LIN {X 0,Y 245.755,Z 1206.562,A -85,B 0,C 180,E1 11861.498,E2 11861.498} C_VEL
LIN {X 0,Y 251.212,Z 1202.888,A -85,B 0,C 180,E1 11857.29,E2 11857.29} C_VEL
LIN {X 0,Y 258.789,Z 1196.828,A -85,B 0,C 180,E1 11852.877,E2 11852.877} C_VEL
LIN {X 0,Y 267.973,Z 1188.669,A -85,B 0,C 180,E1 11848.76,E2 11848.76} C_VEL
LIN {X 0,Y 278.335,Z 1179.083,A -85,B 0,C 180,E1 11845.169,E2 11845.169} C_VEL
LIN {X 0,Y 289.084,Z 1169.149,A -85,B 0,C 180,E1 11842.216,E2 11842.216} C_VEL
LIN {X 0,Y 274.237,Z 1186.667,A -85,B 0,C 180,E1 11838.684,E2 11838.684} C_VEL
LIN {X 0,Y 269.596,Z 1192.92,A -85,B 0,C 180,E1 11837.251,E2 11837.251} C_VEL
LIN {X 0,Y 262.948,Z 1209.699,A -85,B 0,C 180,E1 11834.368,E2 11834.368} C_VEL
LIN {X 0,Y 256.592,Z 1224.704,A -85,B 0,C 180,E1 11831.19,E2 11831.19} C_VEL
LIN {X 0,Y 250.584,Z 1238.42,A -85,B 0,C 180,E1 11827.626,E2 11827.626} C_VEL
LIN {X 0,Y 244.864,Z 1251.431,A -85,B 0,C 180,E1 11823.454,E2 11823.454} C_VEL
LIN {X 0,Y 240.269,Z 1262.385,A -85,B 0,C 180,E1 11819.086,E2 11819.086} C_VEL
LIN {X 0,Y 236.737,Z 1271.709,A -85,B 0,C 180,E1 11814.451,E2 11814.451} C_VEL
LIN {X 0,Y 234.239,Z 1279.61,A -85,B 0,C 180,E1 11809.449,E2 11809.449} C_VEL
LIN {X 0,Y 232.909,Z 1285.561,A -85,B 0,C 180,E1 11804.419,E2 11804.419} C_VEL
LIN {X 0,Y 232.494,Z 1289.538,A -85,B 0,C 180,E1 11799.656,E2 11799.656} C_VEL
LIN {X 0,Y 232.55,Z 1291.91,A -85,B 0,C 180,E1 11795.181,E2 11795.181} C_VEL
LIN {X 0,Y 232.656,Z 1292.783,A -85,B 0,C 180,E1 11791.232,E2 11791.232} C_VEL
LIN {X 0,Y 232.611,Z 1292.569,A -85,B 0,C 180,E1 11787.044,E2 11787.044} C_VEL
LIN {X 0,Y 232.476,Z 1291.001,A -85,B 0,C 180,E1 11782.836,E2 11782.836} C_VEL
LIN {X 0,Y 232.564,Z 1287.833,A -85,B 0,C 180,E1 11778.092,E2 11778.092} C_VEL
LIN {X 0,Y 233.279,Z 1283.097,A -85,B 0,C 180,E1 11773.313,E2 11773.313} C_VEL
LIN {X 0,Y 235.041,Z 1276.237,A -85,B 0,C 180,E1 11768.28,E2 11768.28} C_VEL
LIN {X 0,Y 237.87,Z 1267.902,A -85,B 0,C 180,E1 11763.542,E2 11763.542} C_VEL
LIN {X 0,Y 241.926,Z 1257.624,A -85,B 0,C 180,E1 11758.896,E2 11758.896} C_VEL
LIN {X 0,Y 246.929,Z 1245.842,A -85,B 0,C 180,E1 11754.619,E2 11754.619} C_VEL
LIN {X 0,Y 252.321,Z 1233.449,A -85,B 0,C 180,E1 11750.947,E2 11750.947} C_VEL
LIN {X 0,Y 258.618,Z 1218.846,A -85,B 0,C 180,E1 11747.425,E2 11747.425} C_VEL
LIN {X 0,Y 265.286,Z 1202.614,A -85,B 0,C 180,E1 11744.268,E2 11744.268} C_VEL
LIN {X 0,Y 271.623,Z 1185.934,A -85,B 0,C 180,E1 11741.649,E2 11741.649} C_VEL
LIN {X 0,Y 277.349,Z 1169.272,A -85,B 0,C 180,E1 11739.515,E2 11739.515} C_VEL
LIN {X 0,Y 283.124,Z 1150.359,A -85,B 0,C 180,E1 11737.565,E2 11737.565} C_VEL
LIN {X 0,Y 288.024,Z 1131.481,A -85,B 0,C 180,E1 11736.019,E2 11736.019} C_VEL
LIN {X 0,Y 292.141,Z 1112.055,A -85,B 0,C 180,E1 11734.776,E2 11734.776} C_VEL
LIN {X 0,Y 295.622,Z 1090.355,A -85,B 0,C 180,E1 11733.771,E2 11733.771} C_VEL
LIN {X 0,Y 297.824,Z 1068.85,A -85,B 0,C 180,E1 11733.095,E2 11733.095} C_VEL
LIN {X 0,Y 300.881,Z 1025.521,A -85,B 0,C 180,E1 11732.117,E2 11732.117} C_VEL
LIN {X 0,Y 303.528,Z 1000.807,A -85,B 0,C 180,E1 11731.837,E2 11731.837} C_VEL
LIN {X 0,Y 305.997,Z 989.84,A -85,B 0,C 180,E1 11731.66,E2 11731.66} C_VEL
LIN {X 0,Y 318.999,Z 964.24,A -85,B 0,C 180,E1 11730.364,E2 11730.364} C_VEL
LIN {X 0,Y 315.803,Z 942.601,A -85,B 0,C 180,E1 11727.022,E2 11727.022} C_VEL
LIN {X 0,Y 315.15,Z 920.536,A -85,B 0,C 180,E1 11723.86,E2 11723.86} C_VEL
LIN {X 0,Y 316.957,Z 896.197,A -85,B 0,C 180,E1 11720.689,E2 11720.689} C_VEL
LIN {X 0,Y 321.01,Z 872.026,A -85,B 0,C 180,E1 11717.866,E2 11717.866} C_VEL
LIN {X 0,Y 322.933,Z 862.716,A -85,B 0,C 180,E1 11716.827,E2 11716.827} C_VEL
LIN {X 0,Y 315.425,Z 847.371,A -85,B 0,C 180,E1 11712.634,E2 11712.634} C_VEL
LIN {X 0,Y 308.32,Z 833.413,A -85,B 0,C 180,E1 11708.391,E2 11708.391} C_VEL
LIN {X 0,Y 302.039,Z 821.447,A -85,B 0,C 180,E1 11704.366,E2 11704.366} C_VEL
LIN {X 0,Y 295.476,Z 809.112,A -85,B 0,C 180,E1 11699.806,E2 11699.806} C_VEL
LIN {X 0,Y 289.595,Z 798.554,A -85,B 0,C 180,E1 11695.445,E2 11695.445} C_VEL
LIN {X 0,Y 285.543,Z 791.156,A -85,B 0,C 180,E1 11692.151,E2 11692.151} C_VEL
LIN {X 0,Y 289.879,Z 787.525,A -85,B 0,C 180,E1 11688.056,E2 11688.056} C_VEL
LIN {X 0,Y 293.724,Z 785.356,A -85,B 0,C 180,E1 11685.208,E2 11685.208} C_VEL
LIN {X 0,Y 295.4,Z 784.737,A -85,B 0,C 180,E1 11684.087,E2 11684.087} C_VEL
LIN {X 0,Y 298.61,Z 791.453,A -85,B 0,C 180,E1 11680.59,E2 11680.59} C_VEL
LIN {X 0,Y 303.9,Z 799.813,A -85,B 0,C 180,E1 11677.359,E2 11677.359} C_VEL
LIN {X 0,Y 310.112,Z 810.178,A -85,B 0,C 180,E1 11674.146,E2 11674.146} C_VEL
LIN {X 0,Y 316.83,Z 822.326,A -85,B 0,C 180,E1 11671.128,E2 11671.128} C_VEL
LIN {X 0,Y 322.139,Z 832.942,A -85,B 0,C 180,E1 11668.972,E2 11668.972} C_VEL
LIN {X 0,Y 306.661,Z 1049.725,A -85,B 0,C 180,E1 11664.3,E2 11664.3} C_VEL
LIN {X 0,Y 304.158,Z 1070.256,A -85,B 0,C 180,E1 11663.577,E2 11663.577} C_VEL
LIN {X 0,Y 300.574,Z 1090.531,A -85,B 0,C 180,E1 11662.568,E2 11662.568} C_VEL
LIN {X 0,Y 296.047,Z 1110.096,A -85,B 0,C 180,E1 11661.275,E2 11661.275} C_VEL
LIN {X 0,Y 290.869,Z 1128.33,A -85,B 0,C 180,E1 11659.739,E2 11659.739} C_VEL
LIN {X 0,Y 284.758,Z 1146.545,A -85,B 0,C 180,E1 11657.804,E2 11657.804} C_VEL
LIN {X 0,Y 278.126,Z 1163.631,A -85,B 0,C 180,E1 11655.527,E2 11655.527} C_VEL
LIN {X 0,Y 271.382,Z 1179.111,A -85,B 0,C 180,E1 11652.967,E2 11652.967} C_VEL
LIN {X 0,Y 264.466,Z 1193.663,A -85,B 0,C 180,E1 11649.993,E2 11649.993} C_VEL
LIN {X 0,Y 257.465,Z 1207.393,A -85,B 0,C 180,E1 11646.497,E2 11646.497} C_VEL
LIN {X 0,Y 250.894,Z 1219.705,A -85,B 0,C 180,E1 11642.546,E2 11642.546} C_VEL
LIN {X 0,Y 245.417,Z 1229.787,A -85,B 0,C 180,E1 11638.467,E2 11638.467} C_VEL
LIN {X 0,Y 240.745,Z 1238.513,A -85,B 0,C 180,E1 11633.977,E2 11633.977} C_VEL
LIN {X 0,Y 237.146,Z 1245.644,A -85,B 0,C 180,E1 11629.189,E2 11629.189} C_VEL
LIN {X 0,Y 234.629,Z 1251.19,A -85,B 0,C 180,E1 11624.057,E2 11624.057} C_VEL
LIN {X 0,Y 233.286,Z 1254.753,A -85,B 0,C 180,E1 11619.123,E2 11619.123} C_VEL
LIN {X 0,Y 232.704,Z 1256.778,A -85,B 0,C 180,E1 11614.188,E2 11614.188} C_VEL
LIN {X 0,Y 232.587,Z 1257.354,A -85,B 0,C 180,E1 11609.506,E2 11609.506} C_VEL
LIN {X 0,Y 232.77,Z 1256.558,A -85,B 0,C 180,E1 11604.824,E2 11604.824} C_VEL
LIN {X 0,Y 233.416,Z 1254.378,A -85,B 0,C 180,E1 11600.133,E2 11600.133} C_VEL
LIN {X 0,Y 234.984,Z 1250.341,A -85,B 0,C 180,E1 11594.955,E2 11594.955} C_VEL
LIN {X 0,Y 237.562,Z 1244.786,A -85,B 0,C 180,E1 11590.066,E2 11590.066} C_VEL
LIN {X 0,Y 241.366,Z 1237.412,A -85,B 0,C 180,E1 11585.266,E2 11585.266} C_VEL
LIN {X 0,Y 246.175,Z 1228.535,A -85,B 0,C 180,E1 11580.83,E2 11580.83} C_VEL
LIN {X 0,Y 252.162,Z 1217.537,A -85,B 0,C 180,E1 11576.553,E2 11576.553} C_VEL
LIN {X 0,Y 258.483,Z 1205.616,A -85,B 0,C 180,E1 11572.883,E2 11572.883} C_VEL
LIN {X 0,Y 265.231,Z 1192.273,A -85,B 0,C 180,E1 11569.578,E2 11569.578} C_VEL
LIN {X 0,Y 272.222,Z 1177.437,A -85,B 0,C 180,E1 11566.618,E2 11566.618} C_VEL
LIN {X 0,Y 279.281,Z 1160.958,A -85,B 0,C 180,E1 11563.977,E2 11563.977} C_VEL
LIN {X 0,Y 285.708,Z 1144.096,A -85,B 0,C 180,E1 11561.805,E2 11561.805} C_VEL
LIN {X 0,Y 291.587,Z 1126.39,A -85,B 0,C 180,E1 11559.968,E2 11559.968} C_VEL
LIN {X 0,Y 297.09,Z 1106.623,A -85,B 0,C 180,E1 11558.356,E2 11558.356} C_VEL
LIN {X 0,Y 301.475,Z 1086.784,A -85,B 0,C 180,E1 11557.11,E2 11557.11} C_VEL
LIN {X 0,Y 302.005,Z 1083.684,A -85,B 0,C 180,E1 11556.935,E2 11556.935} C_VEL
LIN {X 0,Y 296.347,Z 1090.87,A -85,B 0,C 180,E1 11556.189,E2 11556.189} C_VEL
LIN {X 0,Y 293.428,Z 1094.102,A -85,B 0,C 180,E1 11555.748,E2 11555.748} C_VEL
LIN {X 0,Y 287.309,Z 1102.337,A -85,B 0,C 180,E1 11555.045,E2 11555.045} C_VEL
LIN {X 0,Y 285.957,Z 1103.878,A -85,B 0,C 180,E1 11554.857,E2 11554.857} C_VEL
LIN {X 0,Y 279.453,Z 1111.591,A -85,B 0,C 180,E1 11553.999,E2 11553.999} C_VEL
LIN {X 0,Y 268.229,Z 1125.113,A -85,B 0,C 180,E1 11552.715,E2 11552.715} C_VEL
LIN {X 0,Y 264.784,Z 1128.644,A -85,B 0,C 180,E1 11552.213,E2 11552.213} C_VEL
LIN {X 0,Y 259.686,Z 1132.965,A -85,B 0,C 180,E1 11551.266,E2 11551.266} C_VEL
LIN {X 0,Y 255.075,Z 1135.823,A -85,B 0,C 180,E1 11550.116,E2 11550.116} C_VEL
LIN {X 0,Y 253.809,Z 1136.519,A -85,B 0,C 180,E1 11549.76,E2 11549.76} C_VEL
LIN {X 0,Y 249.389,Z 1139.988,A -85,B 0,C 180,E1 11548.758,E2 11548.758} C_VEL
LIN {X 0,Y 245.814,Z 1141.922,A -85,B 0,C 180,E1 11547.627,E2 11547.627} C_VEL
LIN {X 0,Y 244.729,Z 1142.395,A -85,B 0,C 180,E1 11547.232,E2 11547.232} C_VEL
LIN {X 0,Y 240.474,Z 1145.51,A -85,B 0,C 180,E1 11546.089,E2 11546.089} C_VEL
LIN {X 0,Y 238.016,Z 1146.572,A -85,B 0,C 180,E1 11545.106,E2 11545.106} C_VEL
LIN {X 0,Y 237.268,Z 1146.582,A -85,B 0,C 180,E1 11544.658,E2 11544.658} C_VEL
LIN {X 0,Y 234.207,Z 1160.293,A -85,B 0,C 180,E1 11541.277,E2 11541.277} C_VEL
LIN {X 0,Y 231.739,Z 1171.635,A -85,B 0,C 180,E1 11537.839,E2 11537.839} C_VEL
LIN {X 0,Y 229.663,Z 1182.256,A -85,B 0,C 180,E1 11533.854,E2 11533.854} C_VEL
LIN {X 0,Y 228.345,Z 1190.868,A -85,B 0,C 180,E1 11529.833,E2 11529.833} C_VEL
LIN {X 0,Y 227.639,Z 1198.409,A -85,B 0,C 180,E1 11525.293,E2 11525.293} C_VEL
LIN {X 0,Y 227.7,Z 1204.054,A -85,B 0,C 180,E1 11520.755,E2 11520.755} C_VEL
LIN {X 0,Y 228.533,Z 1208.064,A -85,B 0,C 180,E1 11515.986,E2 11515.986} C_VEL
LIN {X 0,Y 230.183,Z 1210.229,A -85,B 0,C 180,E1 11511.508,E2 11511.508} C_VEL
LIN {X 0,Y 233.338,Z 1210.736,A -85,B 0,C 180,E1 11506.369,E2 11506.369} C_VEL
LIN {X 0,Y 237.731,Z 1209.285,A -85,B 0,C 180,E1 11501.613,E2 11501.613} C_VEL
LIN {X 0,Y 243.617,Z 1206.041,A -85,B 0,C 180,E1 11497.052,E2 11497.052} C_VEL
LIN {X 0,Y 251.038,Z 1200.995,A -85,B 0,C 180,E1 11492.74,E2 11492.74} C_VEL
LIN {X 0,Y 259.977,Z 1194.181,A -85,B 0,C 180,E1 11488.722,E2 11488.722} C_VEL
LIN {X 0,Y 271.054,Z 1185.201,A -85,B 0,C 180,E1 11484.869,E2 11484.869} C_VEL
LIN {X 0,Y 279.911,Z 1178.049,A -85,B 0,C 180,E1 11482.384,E2 11482.384} C_VEL
LIN {X 0,Y 266.206,Z 1192.836,A -85,B 0,C 180,E1 11479.022,E2 11479.022} C_VEL
LIN {X 0,Y 261.249,Z 1199.161,A -85,B 0,C 180,E1 11477.456,E2 11477.456} C_VEL
LIN {X 0,Y 254.581,Z 1214.76,A -85,B 0,C 180,E1 11474.513,E2 11474.513} C_VEL
LIN {X 0,Y 247.632,Z 1230.01,A -85,B 0,C 180,E1 11470.971,E2 11470.971} C_VEL
LIN {X 0,Y 241.173,Z 1243.865,A -85,B 0,C 180,E1 11466.953,E2 11466.953} C_VEL
LIN {X 0,Y 235.919,Z 1255.286,A -85,B 0,C 180,E1 11462.854,E2 11462.854} C_VEL
LIN {X 0,Y 231.476,Z 1265.398,A -85,B 0,C 180,E1 11458.37,E2 11458.37} C_VEL
LIN {X 0,Y 227.935,Z 1274.476,A -85,B 0,C 180,E1 11453.254,E2 11453.254} C_VEL
LIN {X 0,Y 225.745,Z 1281.555,A -85,B 0,C 180,E1 11448.063,E2 11448.063} C_VEL
LIN {X 0,Y 224.733,Z 1286.663,A -85,B 0,C 180,E1 11443.007,E2 11443.007} C_VEL
LIN {X 0,Y 224.499,Z 1290.151,A -85,B 0,C 180,E1 11437.937,E2 11437.937} C_VEL
LIN {X 0,Y 224.622,Z 1291.82,A -85,B 0,C 180,E1 11433.574,E2 11433.574} C_VEL
LIN {X 0,Y 224.683,Z 1292.221,A -85,B 0,C 180,E1 11429.236,E2 11429.236} C_VEL
LIN {X 0,Y 224.57,Z 1291.442,A -85,B 0,C 180,E1 11425.148,E2 11425.148} C_VEL
LIN {X 0,Y 224.475,Z 1289.247,A -85,B 0,C 180,E1 11420.515,E2 11420.515} C_VEL
LIN {X 0,Y 224.833,Z 1285.436,A -85,B 0,C 180,E1 11415.581,E2 11415.581} C_VEL
LIN {X 0,Y 226.141,Z 1279.594,A -85,B 0,C 180,E1 11410.366,E2 11410.366} C_VEL
LIN {X 0,Y 228.519,Z 1272.303,A -85,B 0,C 180,E1 11405.44,E2 11405.44} C_VEL
LIN {X 0,Y 232.281,Z 1262.786,A -85,B 0,C 180,E1 11400.401,E2 11400.401} C_VEL
LIN {X 0,Y 237.232,Z 1251.545,A -85,B 0,C 180,E1 11395.697,E2 11395.697} C_VEL
LIN {X 0,Y 242.909,Z 1239.257,A -85,B 0,C 180,E1 11391.573,E2 11391.573} C_VEL
LIN {X 0,Y 249.126,Z 1225.826,A -85,B 0,C 180,E1 11387.915,E2 11387.915} C_VEL
LIN {X 0,Y 256.065,Z 1210.193,A -85,B 0,C 180,E1 11384.479,E2 11384.479} C_VEL
LIN {X 0,Y 263.051,Z 1193.366,A -85,B 0,C 180,E1 11381.515,E2 11381.515} C_VEL
LIN {X 0,Y 269.639,Z 1175.901,A -85,B 0,C 180,E1 11379.045,E2 11379.045} C_VEL
LIN {X 0,Y 275.69,Z 1157.961,A -85,B 0,C 180,E1 11377.016,E2 11377.016} C_VEL
LIN {X 0,Y 281.267,Z 1138.742,A -85,B 0,C 180,E1 11375.281,E2 11375.281} C_VEL
LIN {X 0,Y 286.067,Z 1118.874,A -85,B 0,C 180,E1 11373.892,E2 11373.892} C_VEL
LIN {X 0,Y 289.705,Z 1099.73,A -85,B 0,C 180,E1 11372.866,E2 11372.866} C_VEL
LIN {X 0,Y 292.638,Z 1078.212,A -85,B 0,C 180,E1 11372.055,E2 11372.055} C_VEL
LIN {X 0,Y 296.419,Z 1028.006,A -85,B 0,C 180,E1 11370.853,E2 11370.853} C_VEL
LIN {X 0,Y 299.151,Z 1002.191,A -85,B 0,C 180,E1 11370.546,E2 11370.546} C_VEL
LIN {X 0,Y 301.455,Z 986.208,A -85,B 0,C 180,E1 11370.504,E2 11370.504} C_VEL
LIN {X 0,Y 312.06,Z 965.62,A -85,B 0,C 180,E1 11369.46,E2 11369.46} C_VEL
LIN {X 0,Y 309.246,Z 943.916,A -85,B 0,C 180,E1 11366.085,E2 11366.085} C_VEL
LIN {X 0,Y 308.93,Z 921.474,A -85,B 0,C 180,E1 11362.853,E2 11362.853} C_VEL
LIN {X 0,Y 311.092,Z 897.155,A -85,B 0,C 180,E1 11359.662,E2 11359.662} C_VEL
LIN {X 0,Y 315.581,Z 872.382,A -85,B 0,C 180,E1 11356.757,E2 11356.757} C_VEL
LIN {X 0,Y 316.739,Z 866.806,A -85,B 0,C 180,E1 11356.128,E2 11356.128} C_VEL
LIN {X 0,Y 309.418,Z 851.782,A -85,B 0,C 180,E1 11351.935,E2 11351.935} C_VEL
LIN {X 0,Y 302.652,Z 838.342,A -85,B 0,C 180,E1 11347.784,E2 11347.784} C_VEL
LIN {X 0,Y 295.798,Z 825.23,A -85,B 0,C 180,E1 11343.294,E2 11343.294} C_VEL
LIN {X 0,Y 289.736,Z 813.938,A -85,B 0,C 180,E1 11339.011,E2 11339.011} C_VEL
LIN {X 0,Y 284.111,Z 803.743,A -85,B 0,C 180,E1 11334.75,E2 11334.75} C_VEL
LIN {X 0,Y 282.771,Z 801.018,A -85,B 0,C 180,E1 11333.503,E2 11333.503} C_VEL
LIN {X 0,Y 283.961,Z 799.112,A -85,B 0,C 180,E1 11331.903,E2 11331.903} C_VEL
LIN {X 0,Y 287.775,Z 795.306,A -85,B 0,C 180,E1 11327.967,E2 11327.967} C_VEL
LIN {X 0,Y 292.798,Z 792.422,A -85,B 0,C 180,E1 11324.146,E2 11324.146} C_VEL
LIN {X 0,Y 297.26,Z 799.603,A -85,B 0,C 180,E1 11320.753,E2 11320.753} C_VEL
LIN {X 0,Y 302.329,Z 807.848,A -85,B 0,C 180,E1 11317.594,E2 11317.594} C_VEL
LIN {X 0,Y 308.804,Z 819.094,A -85,B 0,C 180,E1 11314.183,E2 11314.183} C_VEL
LIN {X 0,Y 315.257,Z 831.409,A -85,B 0,C 180,E1 11311.23,E2 11311.23} C_VEL
LIN {X 0,Y 317.829,Z 836.982,A -85,B 0,C 180,E1 11310.13,E2 11310.13} C_VEL
LIN {X 0,Y 302.072,Z 1050.253,A -85,B 0,C 180,E1 11305.53,E2 11305.53} C_VEL
LIN {X 0,Y 299.478,Z 1070.877,A -85,B 0,C 180,E1 11304.803,E2 11304.803} C_VEL
LIN {X 0,Y 295.813,Z 1090.993,A -85,B 0,C 180,E1 11303.803,E2 11303.803} C_VEL
LIN {X 0,Y 291.448,Z 1109.477,A -85,B 0,C 180,E1 11302.594,E2 11302.594} C_VEL
LIN {X 0,Y 286.059,Z 1128.048,A -85,B 0,C 180,E1 11301.049,E2 11301.049} C_VEL
LIN {X 0,Y 279.744,Z 1146.295,A -85,B 0,C 180,E1 11299.122,E2 11299.122} C_VEL
LIN {X 0,Y 273.079,Z 1162.967,A -85,B 0,C 180,E1 11296.916,E2 11296.916} C_VEL
LIN {X 0,Y 266.054,Z 1178.641,A -85,B 0,C 180,E1 11294.346,E2 11294.346} C_VEL
LIN {X 0,Y 258.801,Z 1193.376,A -85,B 0,C 180,E1 11291.348,E2 11291.348} C_VEL
LIN {X 0,Y 251.787,Z 1206.637,A -85,B 0,C 180,E1 11287.988,E2 11287.988} C_VEL
LIN {X 0,Y 245.189,Z 1218.485,A -85,B 0,C 180,E1 11284.245,E2 11284.245} C_VEL
LIN {X 0,Y 239.22,Z 1228.924,A -85,B 0,C 180,E1 11280.095,E2 11280.095} C_VEL
LIN {X 0,Y 233.877,Z 1238.265,A -85,B 0,C 180,E1 11275.309,E2 11275.309} C_VEL
LIN {X 0,Y 229.869,Z 1245.584,A -85,B 0,C 180,E1 11270.362,E2 11270.362} C_VEL
LIN {X 0,Y 227.139,Z 1251.083,A -85,B 0,C 180,E1 11265.313,E2 11265.313} C_VEL
LIN {X 0,Y 225.519,Z 1254.938,A -85,B 0,C 180,E1 11260.177,E2 11260.177} C_VEL
LIN {X 0,Y 224.795,Z 1257.199,A -85,B 0,C 180,E1 11255.102,E2 11255.102} C_VEL
LIN {X 0,Y 224.614,Z 1257.974,A -85,B 0,C 180,E1 11250.254,E2 11250.254} C_VEL
LIN {X 0,Y 224.749,Z 1257.356,A -85,B 0,C 180,E1 11245.406,E2 11245.406} C_VEL
LIN {X 0,Y 225.409,Z 1255.288,A -85,B 0,C 180,E1 11240.295,E2 11240.295} C_VEL
LIN {X 0,Y 226.899,Z 1251.677,A -85,B 0,C 180,E1 11235.191,E2 11235.191} C_VEL
LIN {X 0,Y 229.493,Z 1246.383,A -85,B 0,C 180,E1 11230.132,E2 11230.132} C_VEL
LIN {X 0,Y 233.349,Z 1239.248,A -85,B 0,C 180,E1 11225.17,E2 11225.17} C_VEL
LIN {X 0,Y 238.253,Z 1230.631,A -85,B 0,C 180,E1 11220.592,E2 11220.592} C_VEL
LIN {X 0,Y 244.021,Z 1220.598,A -85,B 0,C 180,E1 11216.415,E2 11216.415} C_VEL
LIN {X 0,Y 250.847,Z 1208.461,A -85,B 0,C 180,E1 11212.421,E2 11212.421} C_VEL
LIN {X 0,Y 257.77,Z 1195.572,A -85,B 0,C 180,E1 11209.039,E2 11209.039} C_VEL
LIN {X 0,Y 264.932,Z 1181.274,A -85,B 0,C 180,E1 11206.018,E2 11206.018} C_VEL
LIN {X 0,Y 272.164,Z 1165.428,A -85,B 0,C 180,E1 11203.33,E2 11203.33} C_VEL
LIN {X 0,Y 279.018,Z 1148.488,A -85,B 0,C 180,E1 11201.032,E2 11201.032} C_VEL
LIN {X 0,Y 285.174,Z 1131.023,A -85,B 0,C 180,E1 11199.132,E2 11199.132} C_VEL
LIN {X 0,Y 290.676,Z 1112.726,A -85,B 0,C 180,E1 11197.545,E2 11197.545} C_VEL
LIN {X 0,Y 293.476,Z 1101.734,A -85,B 0,C 180,E1 11196.746,E2 11196.746} C_VEL
LIN {X 0,Y 287.29,Z 1109.159,A -85,B 0,C 180,E1 11196.028,E2 11196.028} C_VEL
LIN {X 0,Y 281.413,Z 1114.592,A -85,B 0,C 180,E1 11195.141,E2 11195.141} C_VEL
LIN {X 0,Y 278.677,Z 1116.83,A -85,B 0,C 180,E1 11194.659,E2 11194.659} C_VEL
LIN {X 0,Y 272.945,Z 1122.529,A -85,B 0,C 180,E1 11193.836,E2 11193.836} C_VEL
LIN {X 0,Y 266.829,Z 1127.206,A -85,B 0,C 180,E1 11192.657,E2 11192.657} C_VEL
LIN {X 0,Y 264.784,Z 1128.644,A -85,B 0,C 180,E1 11192.213,E2 11192.213} C_VEL
LIN {X 0,Y 248.595,Z 1143.852,A -85,B 0,C 180,E1 11189.563,E2 11189.563} C_VEL
LIN {X 0,Y 242.304,Z 1148.962,A -85,B 0,C 180,E1 11188.267,E2 11188.267} C_VEL
LIN {X 0,Y 237.762,Z 1152.003,A -85,B 0,C 180,E1 11187.012,E2 11187.012} C_VEL
LIN {X 0,Y 234.032,Z 1153.609,A -85,B 0,C 180,E1 11185.564,E2 11185.564} C_VEL
LIN {X 0,Y 230.264,Z 1156.037,A -85,B 0,C 180,E1 11184.363,E2 11184.363} C_VEL
LIN {X 0,Y 227.939,Z 1156.895,A -85,B 0,C 180,E1 11183.253,E2 11183.253} C_VEL
LIN {X 0,Y 227.443,Z 1156.889,A -85,B 0,C 180,E1 11182.896,E2 11182.896} C_VEL
LIN {X 0,Y 224.582,Z 1169.354,A -85,B 0,C 180,E1 11179.236,E2 11179.236} C_VEL
LIN {X 0,Y 222.224,Z 1180.722,A -85,B 0,C 180,E1 11175.128,E2 11175.128} C_VEL
LIN {X 0,Y 220.675,Z 1189.9,A -85,B 0,C 180,E1 11170.971,E2 11170.971} C_VEL
LIN {X 0,Y 219.784,Z 1198.079,A -85,B 0,C 180,E1 11166.269,E2 11166.269} C_VEL
LIN {X 0,Y 219.688,Z 1203.942,A -85,B 0,C 180,E1 11161.826,E2 11161.826} C_VEL
LIN {X 0,Y 220.396,Z 1208.645,A -85,B 0,C 180,E1 11156.88,E2 11156.88} C_VEL
LIN {X 0,Y 221.938,Z 1211.401,A -85,B 0,C 180,E1 11152.233,E2 11152.233} C_VEL
LIN {X 0,Y 224.856,Z 1212.645,A -85,B 0,C 180,E1 11147.154,E2 11147.154} C_VEL
LIN {X 0,Y 229.413,Z 1211.937,A -85,B 0,C 180,E1 11141.975,E2 11141.975} C_VEL
LIN {X 0,Y 235.33,Z 1209.441,A -85,B 0,C 180,E1 11137.255,E2 11137.255} C_VEL
LIN {X 0,Y 242.832,Z 1205.233,A -85,B 0,C 180,E1 11132.804,E2 11132.804} C_VEL
LIN {X 0,Y 252.404,Z 1199.012,A -85,B 0,C 180,E1 11128.474,E2 11128.474} C_VEL
LIN {X 0,Y 263.734,Z 1191.052,A -85,B 0,C 180,E1 11124.547,E2 11124.547} C_VEL
LIN {X 0,Y 270.68,Z 1186.09,A -85,B 0,C 180,E1 11122.579,E2 11122.579} C_VEL
LIN {X 0,Y 255.559,Z 1201.341,A -85,B 0,C 180,E1 11118.609,E2 11118.609} C_VEL
LIN {X 0,Y 253.29,Z 1204.034,A -85,B 0,C 180,E1 11117.851,E2 11117.851} C_VEL
LIN {X 0,Y 246.121,Z 1219.662,A -85,B 0,C 180,E1 11114.654,E2 11114.654} C_VEL
LIN {X 0,Y 239.159,Z 1233.99,A -85,B 0,C 180,E1 11111.025,E2 11111.025} C_VEL
LIN {X 0,Y 232.795,Z 1246.848,A -85,B 0,C 180,E1 11106.964,E2 11106.964} C_VEL
LIN {X 0,Y 227.221,Z 1258.223,A -85,B 0,C 180,E1 11102.47,E2 11102.47} C_VEL
LIN {X 0,Y 222.879,Z 1267.655,A -85,B 0,C 180,E1 11097.812,E2 11097.812} C_VEL
LIN {X 0,Y 219.465,Z 1276.134,A -85,B 0,C 180,E1 11092.502,E2 11092.502} C_VEL
LIN {X 0,Y 217.521,Z 1282.414,A -85,B 0,C 180,E1 11087.385,E2 11087.385} C_VEL
LIN {X 0,Y 216.654,Z 1287.055,A -85,B 0,C 180,E1 11082.258,E2 11082.258} C_VEL
LIN {X 0,Y 216.525,Z 1290.031,A -85,B 0,C 180,E1 11077.163,E2 11077.163} C_VEL
LIN {X 0,Y 216.677,Z 1291.463,A -85,B 0,C 180,E1 11072.381,E2 11072.381} C_VEL
LIN {X 0,Y 216.694,Z 1291.538,A -85,B 0,C 180,E1 11068.415,E2 11068.415} C_VEL
LIN {X 0,Y 216.545,Z 1290.509,A -85,B 0,C 180,E1 11063.905,E2 11063.905} C_VEL
LIN {X 0,Y 216.522,Z 1287.938,A -85,B 0,C 180,E1 11059.088,E2 11059.088} C_VEL
LIN {X 0,Y 217.172,Z 1283.472,A -85,B 0,C 180,E1 11053.691,E2 11053.691} C_VEL
LIN {X 0,Y 218.822,Z 1277.583,A -85,B 0,C 180,E1 11048.56,E2 11048.56} C_VEL
LIN {X 0,Y 221.688,Z 1269.965,A -85,B 0,C 180,E1 11043.481,E2 11043.481} C_VEL
LIN {X 0,Y 225.887,Z 1260.408,A -85,B 0,C 180,E1 11038.514,E2 11038.514} C_VEL
LIN {X 0,Y 231.114,Z 1249.411,A -85,B 0,C 180,E1 11033.96,E2 11033.96} C_VEL
LIN {X 0,Y 237.173,Z 1237.034,A -85,B 0,C 180,E1 11029.835,E2 11029.835} C_VEL
LIN {X 0,Y 244.095,Z 1222.822,A -85,B 0,C 180,E1 11026.03,E2 11026.03} C_VEL
LIN {X 0,Y 250.929,Z 1208.145,A -85,B 0,C 180,E1 11022.849,E2 11022.849} C_VEL
LIN {X 0,Y 258.185,Z 1191.463,A -85,B 0,C 180,E1 11019.936,E2 11019.936} C_VEL
LIN {X 0,Y 265.137,Z 1173.722,A -85,B 0,C 180,E1 11017.458,E2 11017.458} C_VEL
LIN {X 0,Y 271.336,Z 1155.84,A -85,B 0,C 180,E1 11015.477,E2 11015.477} C_VEL
LIN {X 0,Y 276.859,Z 1137.34,A -85,B 0,C 180,E1 11013.838,E2 11013.838} C_VEL
LIN {X 0,Y 281.765,Z 1117.546,A -85,B 0,C 180,E1 11012.473,E2 11012.473} C_VEL
LIN {X 0,Y 285.557,Z 1098,A -85,B 0,C 180,E1 11011.447,E2 11011.447} C_VEL
LIN {X 0,Y 288.522,Z 1077.053,A -85,B 0,C 180,E1 11010.685,E2 11010.685} C_VEL
LIN {X 0,Y 292.421,Z 1027.207,A -85,B 0,C 180,E1 11009.501,E2 11009.501} C_VEL
LIN {X 0,Y 295.203,Z 1001.467,A -85,B 0,C 180,E1 11009.21,E2 11009.21} C_VEL
LIN {X 0,Y 298.349,Z 980.02,A -85,B 0,C 180,E1 11009.191,E2 11009.191} C_VEL
LIN {X 0,Y 305.184,Z 966.967,A -85,B 0,C 180,E1 11008.528,E2 11008.528} C_VEL
LIN {X 0,Y 302.698,Z 944.459,A -85,B 0,C 180,E1 11005.011,E2 11005.011} C_VEL
LIN {X 0,Y 302.828,Z 921.579,A -85,B 0,C 180,E1 11001.702,E2 11001.702} C_VEL
LIN {X 0,Y 305.389,Z 897.359,A -85,B 0,C 180,E1 10998.516,E2 10998.516} C_VEL
LIN {X 0,Y 310.452,Z 871.627,A -85,B 0,C 180,E1 10995.504,E2 10995.504} C_VEL
LIN {X 0,Y 310.409,Z 870.542,A -85,B 0,C 180,E1 10995.315,E2 10995.315} C_VEL
LIN {X 0,Y 303.091,Z 855.47,A -85,B 0,C 180,E1 10991.03,E2 10991.03} C_VEL
LIN {X 0,Y 296.007,Z 841.466,A -85,B 0,C 180,E1 10986.594,E2 10986.594} C_VEL
LIN {X 0,Y 289.742,Z 829.447,A -85,B 0,C 180,E1 10982.373,E2 10982.373} C_VEL
LIN {X 0,Y 283.201,Z 817.126,A -85,B 0,C 180,E1 10977.571,E2 10977.571} C_VEL
LIN {X 0,Y 280.57,Z 812.077,A -85,B 0,C 180,E1 10975.4,E2 10975.4} C_VEL
LIN {X 0,Y 281.665,Z 809.646,A -85,B 0,C 180,E1 10973.579,E2 10973.579} C_VEL
LIN {X 0,Y 282.321,Z 808.421,A -85,B 0,C 180,E1 10972.675,E2 10972.675} C_VEL
LIN {X 0,Y 284.364,Z 805.526,A -85,B 0,C 180,E1 10970.283,E2 10970.283} C_VEL
LIN {X 0,Y 289.692,Z 801.488,A -85,B 0,C 180,E1 10965.611,E2 10965.611} C_VEL
LIN {X 0,Y 291.684,Z 800.728,A -85,B 0,C 180,E1 10964.185,E2 10964.185} C_VEL
LIN {X 0,Y 296.053,Z 807.925,A -85,B 0,C 180,E1 10960.825,E2 10960.825} C_VEL
LIN {X 0,Y 300.914,Z 816.19,A -85,B 0,C 180,E1 10957.741,E2 10957.741} C_VEL
LIN {X 0,Y 307.095,Z 827.439,A -85,B 0,C 180,E1 10954.409,E2 10954.409} C_VEL
LIN {X 0,Y 313.612,Z 840.434,A -85,B 0,C 180,E1 10951.361,E2 10951.361} C_VEL
LIN {X 0,Y 299.561,Z 1026.455,A -85,B 0,C 180,E1 10947.372,E2 10947.372} C_VEL
LIN {X 0,Y 297.181,Z 1055.167,A -85,B 0,C 180,E1 10946.671,E2 10946.671} C_VEL
LIN {X 0,Y 294.185,Z 1076.304,A -85,B 0,C 180,E1 10945.865,E2 10945.865} C_VEL
LIN {X 0,Y 289.917,Z 1097.326,A -85,B 0,C 180,E1 10944.734,E2 10944.734} C_VEL
LIN {X 0,Y 284.649,Z 1117.223,A -85,B 0,C 180,E1 10943.31,E2 10943.31} C_VEL
LIN {X 0,Y 278.772,Z 1135.395,A -85,B 0,C 180,E1 10941.647,E2 10941.647} C_VEL
LIN {X 0,Y 272.202,Z 1152.766,A -85,B 0,C 180,E1 10939.656,E2 10939.656} C_VEL
LIN {X 0,Y 264.731,Z 1170.047,A -85,B 0,C 180,E1 10937.168,E2 10937.168} C_VEL
LIN {X 0,Y 257.019,Z 1185.941,A -85,B 0,C 180,E1 10934.291,E2 10934.291} C_VEL
LIN {X 0,Y 249.506,Z 1200.082,A -85,B 0,C 180,E1 10931.086,E2 10931.086} C_VEL
LIN {X 0,Y 242.512,Z 1212.421,A -85,B 0,C 180,E1 10927.602,E2 10927.602} C_VEL
LIN {X 0,Y 235.623,Z 1223.997,A -85,B 0,C 180,E1 10923.479,E2 10923.479} C_VEL
LIN {X 0,Y 229.483,Z 1234.081,A -85,B 0,C 180,E1 10918.864,E2 10918.864} C_VEL
LIN {X 0,Y 224.49,Z 1242.394,A -85,B 0,C 180,E1 10913.909,E2 10913.909} C_VEL
LIN {X 0,Y 220.827,Z 1248.88,A -85,B 0,C 180,E1 10908.751,E2 10908.751} C_VEL
LIN {X 0,Y 218.458,Z 1253.62,A -85,B 0,C 180,E1 10903.497,E2 10903.497} C_VEL
LIN {X 0,Y 217.174,Z 1256.767,A -85,B 0,C 180,E1 10898.167,E2 10898.167} C_VEL
LIN {X 0,Y 216.701,Z 1258.316,A -85,B 0,C 180,E1 10893.173,E2 10893.173} C_VEL
LIN {X 0,Y 216.64,Z 1258.486,A -85,B 0,C 180,E1 10888.412,E2 10888.412} C_VEL
LIN {X 0,Y 216.956,Z 1257.439,A -85,B 0,C 180,E1 10883.383,E2 10883.383} C_VEL
LIN {X 0,Y 217.954,Z 1254.857,A -85,B 0,C 180,E1 10878.085,E2 10878.085} C_VEL
LIN {X 0,Y 220.082,Z 1250.369,A -85,B 0,C 180,E1 10872.551,E2 10872.551} C_VEL
LIN {X 0,Y 223.393,Z 1244.335,A -85,B 0,C 180,E1 10867.36,E2 10867.36} C_VEL
LIN {X 0,Y 228.037,Z 1236.501,A -85,B 0,C 180,E1 10862.339,E2 10862.339} C_VEL
LIN {X 0,Y 233.806,Z 1227.021,A -85,B 0,C 180,E1 10857.685,E2 10857.685} C_VEL
LIN {X 0,Y 240.385,Z 1216.103,A -85,B 0,C 180,E1 10853.501,E2 10853.501} C_VEL
LIN {X 0,Y 247.568,Z 1203.716,A -85,B 0,C 180,E1 10849.743,E2 10849.743} C_VEL
LIN {X 0,Y 254.723,Z 1190.653,A -85,B 0,C 180,E1 10846.567,E2 10846.567} C_VEL
LIN {X 0,Y 262.361,Z 1175.401,A -85,B 0,C 180,E1 10843.606,E2 10843.606} C_VEL
LIN {X 0,Y 269.499,Z 1159.55,A -85,B 0,C 180,E1 10841.136,E2 10841.136} C_VEL
LIN {X 0,Y 276.154,Z 1142.924,A -85,B 0,C 180,E1 10839.05,E2 10839.05} C_VEL
LIN {X 0,Y 282.482,Z 1124.618,A -85,B 0,C 180,E1 10837.211,E2 10837.211} C_VEL
LIN {X 0,Y 284.393,Z 1118.317,A -85,B 0,C 180,E1 10836.643,E2 10836.643} C_VEL
LIN {X 0,Y 279.173,Z 1122.52,A -85,B 0,C 180,E1 10835.844,E2 10835.844} C_VEL
LIN {X 0,Y 272.497,Z 1128.728,A -85,B 0,C 180,E1 10834.918,E2 10834.918} C_VEL
LIN {X 0,Y 266.186,Z 1133.264,A -85,B 0,C 180,E1 10833.775,E2 10833.775} C_VEL
LIN {X 0,Y 263.831,Z 1134.97,A -85,B 0,C 180,E1 10833.334,E2 10833.334} C_VEL
LIN {X 0,Y 257.369,Z 1139.923,A -85,B 0,C 180,E1 10832.121,E2 10832.121} C_VEL
LIN {X 0,Y 251.893,Z 1143.176,A -85,B 0,C 180,E1 10830.801,E2 10830.801} C_VEL
LIN {X 0,Y 246.751,Z 1146.696,A -85,B 0,C 180,E1 10829.628,E2 10829.628} C_VEL
LIN {X 0,Y 242.304,Z 1148.962,A -85,B 0,C 180,E1 10828.267,E2 10828.267} C_VEL
LIN {X 0,Y 226.363,Z 1161.768,A -85,B 0,C 180,E1 10824.567,E2 10824.567} C_VEL
LIN {X 0,Y 221.381,Z 1165.109,A -85,B 0,C 180,E1 10822.938,E2 10822.938} C_VEL
LIN {X 0,Y 220.813,Z 1165.424,A -85,B 0,C 180,E1 10822.71,E2 10822.71} C_VEL
LIN {X 0,Y 218.084,Z 1166.441,A -85,B 0,C 180,E1 10821.236,E2 10821.236} C_VEL
LIN {X 0,Y 217.588,Z 1166.582,A -85,B 0,C 180,E1 10820.793,E2 10820.793} C_VEL
LIN {X 0,Y 214.94,Z 1178.633,A -85,B 0,C 180,E1 10816.608,E2 10816.608} C_VEL
LIN {X 0,Y 213.056,Z 1188.702,A -85,B 0,C 180,E1 10812.192,E2 10812.192} C_VEL
LIN {X 0,Y 211.988,Z 1197.104,A -85,B 0,C 180,E1 10807.589,E2 10807.589} C_VEL
LIN {X 0,Y 211.704,Z 1203.925,A -85,B 0,C 180,E1 10802.708,E2 10802.708} C_VEL
LIN {X 0,Y 212.262,Z 1208.996,A -85,B 0,C 180,E1 10797.841,E2 10797.841} C_VEL
LIN {X 0,Y 213.797,Z 1212.479,A -85,B 0,C 180,E1 10792.746,E2 10792.746} C_VEL
LIN {X 0,Y 216.529,Z 1214.297,A -85,B 0,C 180,E1 10787.737,E2 10787.737} C_VEL
LIN {X 0,Y 221.31,Z 1214.32,A -85,B 0,C 180,E1 10782.109,E2 10782.109} C_VEL
LIN {X 0,Y 228.036,Z 1212.232,A -85,B 0,C 180,E1 10776.758,E2 10776.758} C_VEL
LIN {X 0,Y 236.73,Z 1208.121,A -85,B 0,C 180,E1 10771.768,E2 10771.768} C_VEL
LIN {X 0,Y 247.91,Z 1201.771,A -85,B 0,C 180,E1 10767.012,E2 10767.012} C_VEL
LIN {X 0,Y 260.62,Z 1193.925,A -85,B 0,C 180,E1 10762.964,E2 10762.964} C_VEL
LIN {X 0,Y 261.257,Z 1193.555,A -85,B 0,C 180,E1 10762.754,E2 10762.754} C_VEL
LIN {X 0,Y 245.963,Z 1207.944,A -85,B 0,C 180,E1 10758.502,E2 10758.502} C_VEL
LIN {X 0,Y 243.729,Z 1211.915,A -85,B 0,C 180,E1 10757.598,E2 10757.598} C_VEL
LIN {X 0,Y 236.963,Z 1225.626,A -85,B 0,C 180,E1 10754.463,E2 10754.463} C_VEL
LIN {X 0,Y 229.624,Z 1239.697,A -85,B 0,C 180,E1 10750.452,E2 10750.452} C_VEL
LIN {X 0,Y 223.027,Z 1252.164,A -85,B 0,C 180,E1 10745.966,E2 10745.966} C_VEL
LIN {X 0,Y 217.729,Z 1262.532,A -85,B 0,C 180,E1 10741.261,E2 10741.261} C_VEL
LIN {X 0,Y 213.508,Z 1271.516,A -85,B 0,C 180,E1 10736.118,E2 10736.118} C_VEL
LIN {X 0,Y 210.555,Z 1279.014,A -85,B 0,C 180,E1 10730.574,E2 10730.574} C_VEL
LIN {X 0,Y 209.04,Z 1284.435,A -85,B 0,C 180,E1 10725.254,E2 10725.254} C_VEL
LIN {X 0,Y 208.532,Z 1288.202,A -85,B 0,C 180,E1 10719.941,E2 10719.941} C_VEL
LIN {X 0,Y 208.613,Z 1290.301,A -85,B 0,C 180,E1 10714.95,E2 10714.95} C_VEL
LIN {X 0,Y 208.731,Z 1291.029,A -85,B 0,C 180,E1 10710.55,E2 10710.55} C_VEL
LIN {X 0,Y 208.64,Z 1290.518,A -85,B 0,C 180,E1 10705.879,E2 10705.879} C_VEL
LIN {X 0,Y 208.492,Z 1288.78,A -85,B 0,C 180,E1 10701.174,E2 10701.174} C_VEL
LIN {X 0,Y 208.792,Z 1285.3,A -85,B 0,C 180,E1 10695.865,E2 10695.865} C_VEL
LIN {X 0,Y 210.114,Z 1279.943,A -85,B 0,C 180,E1 10690.255,E2 10690.255} C_VEL
LIN {X 0,Y 212.622,Z 1273.162,A -85,B 0,C 180,E1 10684.963,E2 10684.963} C_VEL
LIN {X 0,Y 216.709,Z 1264.059,A -85,B 0,C 180,E1 10679.503,E2 10679.503} C_VEL
LIN {X 0,Y 222.061,Z 1253.329,A -85,B 0,C 180,E1 10674.492,E2 10674.492} C_VEL
LIN {X 0,Y 228.458,Z 1241.04,A -85,B 0,C 180,E1 10669.959,E2 10669.959} C_VEL
LIN {X 0,Y 235.174,Z 1228.078,A -85,B 0,C 180,E1 10666.133,E2 10666.133} C_VEL
LIN {X 0,Y 242.532,Z 1213.328,A -85,B 0,C 180,E1 10662.62,E2 10662.62} C_VEL
LIN {X 0,Y 250.147,Z 1197.062,A -85,B 0,C 180,E1 10659.519,E2 10659.519} C_VEL
LIN {X 0,Y 257.231,Z 1180.542,A -85,B 0,C 180,E1 10656.988,E2 10656.988} C_VEL
LIN {X 0,Y 264.168,Z 1162.483,A -85,B 0,C 180,E1 10654.784,E2 10654.784} C_VEL
LIN {X 0,Y 270.657,Z 1142.775,A -85,B 0,C 180,E1 10652.891,E2 10652.891} C_VEL
LIN {X 0,Y 276.021,Z 1123.186,A -85,B 0,C 180,E1 10651.441,E2 10651.441} C_VEL
LIN {X 0,Y 280.193,Z 1104.197,A -85,B 0,C 180,E1 10650.371,E2 10650.371} C_VEL
LIN {X 0,Y 283.523,Z 1083.688,A -85,B 0,C 180,E1 10649.511,E2 10649.511} C_VEL
LIN {X 0,Y 285.869,Z 1061.14,A -85,B 0,C 180,E1 10648.885,E2 10648.885} C_VEL
LIN {X 0,Y 288.605,Z 1026.263,A -85,B 0,C 180,E1 10648.109,E2 10648.109} C_VEL
LIN {X 0,Y 291.428,Z 1000.677,A -85,B 0,C 180,E1 10647.838,E2 10647.838} C_VEL
LIN {X 0,Y 295.062,Z 975.189,A -85,B 0,C 180,E1 10647.87,E2 10647.87} C_VEL
LIN {X 0,Y 295.703,Z 973.327,A -85,B 0,C 180,E1 10647.848,E2 10647.848} C_VEL
LIN {X 0,Y 298.321,Z 968.249,A -85,B 0,C 180,E1 10647.584,E2 10647.584} C_VEL
LIN {X 0,Y 296.225,Z 945.529,A -85,B 0,C 180,E1 10643.999,E2 10643.999} C_VEL
LIN {X 0,Y 296.741,Z 922.305,A -85,B 0,C 180,E1 10640.616,E2 10640.616} C_VEL
LIN {X 0,Y 299.836,Z 896.845,A -85,B 0,C 180,E1 10637.264,E2 10637.264} C_VEL
LIN {X 0,Y 304.302,Z 874.838,A -85,B 0,C 180,E1 10634.655,E2 10634.655} C_VEL
LIN {X 0,Y 297.018,Z 859.748,A -85,B 0,C 180,E1 10630.277,E2 10630.277} C_VEL
LIN {X 0,Y 289.963,Z 845.713,A -85,B 0,C 180,E1 10625.739,E2 10625.739} C_VEL
LIN {X 0,Y 283.707,Z 833.722,A -85,B 0,C 180,E1 10621.413,E2 10621.413} C_VEL
LIN {X 0,Y 278.585,Z 823.764,A -85,B 0,C 180,E1 10617.428,E2 10617.428} C_VEL
LIN {X 0,Y 279.618,Z 820.316,A -85,B 0,C 180,E1 10615.231,E2 10615.231} C_VEL
LIN {X 0,Y 281.631,Z 816.122,A -85,B 0,C 180,E1 10612.246,E2 10612.246} C_VEL
LIN {X 0,Y 283.763,Z 813.228,A -85,B 0,C 180,E1 10609.852,E2 10609.852} C_VEL
LIN {X 0,Y 288.999,Z 809.367,A -85,B 0,C 180,E1 10605.37,E2 10605.37} C_VEL
LIN {X 0,Y 290.45,Z 808.928,A -85,B 0,C 180,E1 10604.321,E2 10604.321} C_VEL
LIN {X 0,Y 294.179,Z 815.186,A -85,B 0,C 180,E1 10601.368,E2 10601.368} C_VEL
LIN {X 0,Y 298.81,Z 823.368,A -85,B 0,C 180,E1 10598.299,E2 10598.299} C_VEL
LIN {X 0,Y 304.59,Z 834.232,A -85,B 0,C 180,E1 10595.05,E2 10595.05} C_VEL
LIN {X 0,Y 309.636,Z 844.747,A -85,B 0,C 180,E1 10592.547,E2 10592.547} C_VEL
LIN {X 0,Y 293.303,Z 1051.587,A -85,B 0,C 180,E1 10588.094,E2 10588.094} C_VEL
LIN {X 0,Y 290.56,Z 1072.062,A -85,B 0,C 180,E1 10587.373,E2 10587.373} C_VEL
LIN {X 0,Y 286.504,Z 1092.892,A -85,B 0,C 180,E1 10586.337,E2 10586.337} C_VEL
LIN {X 0,Y 281.347,Z 1112.963,A -85,B 0,C 180,E1 10584.998,E2 10584.998} C_VEL
LIN {X 0,Y 275.648,Z 1130.995,A -85,B 0,C 180,E1 10583.459,E2 10583.459} C_VEL
LIN {X 0,Y 269.196,Z 1148.348,A -85,B 0,C 180,E1 10581.599,E2 10581.599} C_VEL
LIN {X 0,Y 261.814,Z 1165.446,A -85,B 0,C 180,E1 10579.292,E2 10579.292} C_VEL
LIN {X 0,Y 254.257,Z 1180.936,A -85,B 0,C 180,E1 10576.676,E2 10576.676} C_VEL
LIN {X 0,Y 246.43,Z 1195.497,A -85,B 0,C 180,E1 10573.609,E2 10573.609} C_VEL
LIN {X 0,Y 238.817,Z 1208.61,A -85,B 0,C 180,E1 10570.146,E2 10570.146} C_VEL
LIN {X 0,Y 231.605,Z 1220.328,A -85,B 0,C 180,E1 10566.258,E2 10566.258} C_VEL
LIN {X 0,Y 225.042,Z 1230.65,A -85,B 0,C 180,E1 10561.917,E2 10561.917} C_VEL
LIN {X 0,Y 219.101,Z 1239.919,A -85,B 0,C 180,E1 10556.857,E2 10556.857} C_VEL
LIN {X 0,Y 214.423,Z 1247.481,A -85,B 0,C 180,E1 10551.327,E2 10551.327} C_VEL
LIN {X 0,Y 211.284,Z 1253.034,A -85,B 0,C 180,E1 10545.647,E2 10545.647} C_VEL
LIN {X 0,Y 209.564,Z 1256.59,A -85,B 0,C 180,E1 10540.167,E2 10540.167} C_VEL
LIN {X 0,Y 208.809,Z 1258.608,A -85,B 0,C 180,E1 10534.668,E2 10534.668} C_VEL
LIN {X 0,Y 208.656,Z 1259.18,A -85,B 0,C 180,E1 10529.45,E2 10529.45} C_VEL
LIN {X 0,Y 208.869,Z 1258.45,A -85,B 0,C 180,E1 10524.505,E2 10524.505} C_VEL
LIN {X 0,Y 209.73,Z 1256.214,A -85,B 0,C 180,E1 10519.006,E2 10519.006} C_VEL
LIN {X 0,Y 211.725,Z 1252.182,A -85,B 0,C 180,E1 10513.256,E2 10513.256} C_VEL
LIN {X 0,Y 214.931,Z 1246.629,A -85,B 0,C 180,E1 10507.863,E2 10507.863} C_VEL
LIN {X 0,Y 219.556,Z 1239.255,A -85,B 0,C 180,E1 10502.615,E2 10502.615} C_VEL
LIN {X 0,Y 225.291,Z 1230.375,A -85,B 0,C 180,E1 10497.82,E2 10497.82} C_VEL
LIN {X 0,Y 232.307,Z 1219.371,A -85,B 0,C 180,E1 10493.253,E2 10493.253} C_VEL
LIN {X 0,Y 239.617,Z 1207.442,A -85,B 0,C 180,E1 10489.386,E2 10489.386} C_VEL
LIN {X 0,Y 247.318,Z 1194.088,A -85,B 0,C 180,E1 10485.943,E2 10485.943} C_VEL
LIN {X 0,Y 255.222,Z 1179.24,A -85,B 0,C 180,E1 10482.895,E2 10482.895} C_VEL
LIN {X 0,Y 263.122,Z 1162.745,A -85,B 0,C 180,E1 10480.199,E2 10480.199} C_VEL
LIN {X 0,Y 270.273,Z 1145.864,A -85,B 0,C 180,E1 10478.002,E2 10478.002} C_VEL
LIN {X 0,Y 275.253,Z 1132.113,A -85,B 0,C 180,E1 10476.501,E2 10476.501} C_VEL
LIN {X 0,Y 267.842,Z 1137.747,A -85,B 0,C 180,E1 10475.354,E2 10475.354} C_VEL
LIN {X 0,Y 263.463,Z 1140.696,A -85,B 0,C 180,E1 10474.559,E2 10474.559} C_VEL
LIN {X 0,Y 256.475,Z 1145.683,A -85,B 0,C 180,E1 10473.346,E2 10473.346} C_VEL
LIN {X 0,Y 250.724,Z 1148.998,A -85,B 0,C 180,E1 10472.032,E2 10472.032} C_VEL
LIN {X 0,Y 244.725,Z 1152.885,A -85,B 0,C 180,E1 10470.711,E2 10470.711} C_VEL
LIN {X 0,Y 240.213,Z 1155.092,A -85,B 0,C 180,E1 10469.418,E2 10469.418} C_VEL
LIN {X 0,Y 234.748,Z 1158.379,A -85,B 0,C 180,E1 10467.939,E2 10467.939} C_VEL
LIN {X 0,Y 231.435,Z 1159.738,A -85,B 0,C 180,E1 10466.7,E2 10466.7} C_VEL
LIN {X 0,Y 227.057,Z 1162.377,A -85,B 0,C 180,E1 10465.287,E2 10465.287} C_VEL
LIN {X 0,Y 223.615,Z 1163.727,A -85,B 0,C 180,E1 10463.73,E2 10463.73} C_VEL
LIN {X 0,Y 220.813,Z 1165.424,A -85,B 0,C 180,E1 10462.71,E2 10462.71} C_VEL
LIN {X 0,Y 216.013,Z 1168.61,A -85,B 0,C 180,E1 10460.825,E2 10460.825} C_VEL
LIN {X 0,Y 210.005,Z 1173.502,A -85,B 0,C 180,E1 10459.024,E2 10459.024} C_VEL
LIN {X 0,Y 207.9,Z 1175.818,A -85,B 0,C 180,E1 10458.321,E2 10458.321} C_VEL
LIN {X 0,Y 207.746,Z 1176.232,A -85,B 0,C 180,E1 10458.166,E2 10458.166} C_VEL
LIN {X 0,Y 205.516,Z 1187.299,A -85,B 0,C 180,E1 10453.505,E2 10453.505} C_VEL
LIN {X 0,Y 204.268,Z 1195.823,A -85,B 0,C 180,E1 10449.012,E2 10449.012} C_VEL
LIN {X 0,Y 203.759,Z 1203.728,A -85,B 0,C 180,E1 10443.658,E2 10443.658} C_VEL
LIN {X 0,Y 204.188,Z 1209.313,A -85,B 0,C 180,E1 10438.598,E2 10438.598} C_VEL
LIN {X 0,Y 205.761,Z 1213.599,A -85,B 0,C 180,E1 10433.023,E2 10433.023} C_VEL
LIN {X 0,Y 208.699,Z 1215.915,A -85,B 0,C 180,E1 10427.55,E2 10427.55} C_VEL
LIN {X 0,Y 213.156,Z 1216.473,A -85,B 0,C 180,E1 10422.249,E2 10422.249} C_VEL
LIN {X 0,Y 219.647,Z 1215.238,A -85,B 0,C 180,E1 10416.954,E2 10416.954} C_VEL
LIN {X 0,Y 228.436,Z 1212.007,A -85,B 0,C 180,E1 10411.79,E2 10411.79} C_VEL
LIN {X 0,Y 239.763,Z 1206.653,A -85,B 0,C 180,E1 10406.887,E2 10406.887} C_VEL
LIN {X 0,Y 251.84,Z 1200.314,A -85,B 0,C 180,E1 10402.942,E2 10402.942} C_VEL
LIN {X 0,Y 237.346,Z 1213.025,A -85,B 0,C 180,E1 10398.716,E2 10398.716} C_VEL
LIN {X 0,Y 229.337,Z 1228.139,A -85,B 0,C 180,E1 10395.067,E2 10395.067} C_VEL
LIN {X 0,Y 222.08,Z 1241.25,A -85,B 0,C 180,E1 10391.098,E2 10391.098} C_VEL
LIN {X 0,Y 215.423,Z 1253.137,A -85,B 0,C 180,E1 10386.588,E2 10386.588} C_VEL
LIN {X 0,Y 209.821,Z 1263.502,A -85,B 0,C 180,E1 10381.614,E2 10381.614} C_VEL
LIN {X 0,Y 205.305,Z 1272.585,A -85,B 0,C 180,E1 10375.997,E2 10375.997} C_VEL
LIN {X 0,Y 202.379,Z 1279.673,A -85,B 0,C 180,E1 10370.234,E2 10370.234} C_VEL
LIN {X 0,Y 200.938,Z 1284.702,A -85,B 0,C 180,E1 10364.702,E2 10364.702} C_VEL
LIN {X 0,Y 200.528,Z 1288.186,A -85,B 0,C 180,E1 10359.163,E2 10359.163} C_VEL
LIN {X 0,Y 200.657,Z 1289.914,A -85,B 0,C 180,E1 10354.288,E2 10354.288} C_VEL
LIN {X 0,Y 200.758,Z 1290.441,A -85,B 0,C 180,E1 10349.716,E2 10349.716} C_VEL
LIN {X 0,Y 200.625,Z 1289.756,A -85,B 0,C 180,E1 10345.141,E2 10345.141} C_VEL
LIN {X 0,Y 200.512,Z 1287.735,A -85,B 0,C 180,E1 10339.95,E2 10339.95} C_VEL
LIN {X 0,Y 200.961,Z 1284.23,A -85,B 0,C 180,E1 10334.712,E2 10334.712} C_VEL
LIN {X 0,Y 202.584,Z 1278.66,A -85,B 0,C 180,E1 10328.876,E2 10328.876} C_VEL
LIN {X 0,Y 205.68,Z 1271.251,A -85,B 0,C 180,E1 10323.123,E2 10323.123} C_VEL
LIN {X 0,Y 210.106,Z 1262.353,A -85,B 0,C 180,E1 10317.794,E2 10317.794} C_VEL
LIN {X 0,Y 215.786,Z 1251.842,A -85,B 0,C 180,E1 10312.841,E2 10312.841} C_VEL
LIN {X 0,Y 222.819,Z 1239.173,A -85,B 0,C 180,E1 10308.149,E2 10308.149} C_VEL
LIN {X 0,Y 230.671,Z 1224.843,A -85,B 0,C 180,E1 10303.986,E2 10303.986} C_VEL
LIN {X 0,Y 238.442,Z 1209.862,A -85,B 0,C 180,E1 10300.538,E2 10300.538} C_VEL
LIN {X 0,Y 246.121,Z 1193.966,A -85,B 0,C 180,E1 10297.612,E2 10297.612} C_VEL
LIN {X 0,Y 253.577,Z 1176.947,A -85,B 0,C 180,E1 10295.1,E2 10295.1} C_VEL
LIN {X 0,Y 260.857,Z 1158.247,A -85,B 0,C 180,E1 10292.923,E2 10292.923} C_VEL
LIN {X 0,Y 267.107,Z 1139.536,A -85,B 0,C 180,E1 10291.205,E2 10291.205} C_VEL
LIN {X 0,Y 272.541,Z 1120.058,A -85,B 0,C 180,E1 10289.817,E2 10289.817} C_VEL
LIN {X 0,Y 276.941,Z 1099.738,A -85,B 0,C 180,E1 10288.722,E2 10288.722} C_VEL
LIN {X 0,Y 280.161,Z 1079.468,A -85,B 0,C 180,E1 10287.96,E2 10287.96} C_VEL
LIN {X 0,Y 282.712,Z 1052.344,A -85,B 0,C 180,E1 10287.258,E2 10287.258} C_VEL
LIN {X 0,Y 285.011,Z 1024.729,A -85,B 0,C 180,E1 10286.669,E2 10286.669} C_VEL
LIN {X 0,Y 288.148,Z 997.331,A -85,B 0,C 180,E1 10286.421,E2 10286.421} C_VEL
LIN {X 0,Y 292.08,Z 969.829,A -85,B 0,C 180,E1 10286.48,E2 10286.48} C_VEL
LIN {X 0,Y 290.641,Z 961.837,A -85,B 0,C 180,E1 10285.359,E2 10285.359} C_VEL
LIN {X 0,Y 289.817,Z 938.688,A -85,B 0,C 180,E1 10281.769,E2 10281.769} C_VEL
LIN {X 0,Y 291.65,Z 913.975,A -85,B 0,C 180,E1 10278.265,E2 10278.265} C_VEL
LIN {X 0,Y 295.862,Z 888.896,A -85,B 0,C 180,E1 10275.083,E2 10275.083} C_VEL
LIN {X 0,Y 298.089,Z 878.819,A -85,B 0,C 180,E1 10273.876,E2 10273.876} C_VEL
LIN {X 0,Y 290.937,Z 864.001,A -85,B 0,C 180,E1 10269.492,E2 10269.492} C_VEL
LIN {X 0,Y 283.904,Z 849.876,A -85,B 0,C 180,E1 10264.848,E2 10264.848} C_VEL
LIN {X 0,Y 277.114,Z 836.767,A -85,B 0,C 180,E1 10260,E2 10260} C_VEL
LIN {X 0,Y 276.92,Z 835.746,A -85,B 0,C 180,E1 10259.379,E2 10259.379} C_VEL
LIN {X 0,Y 277.975,Z 830.64,A -85,B 0,C 180,E1 10256.391,E2 10256.391} C_VEL
LIN {X 0,Y 279.297,Z 826.986,A -85,B 0,C 180,E1 10254.041,E2 10254.041} C_VEL
LIN {X 0,Y 281.122,Z 823.595,A -85,B 0,C 180,E1 10251.615,E2 10251.615} C_VEL
LIN {X 0,Y 283.176,Z 820.942,A -85,B 0,C 180,E1 10249.42,E2 10249.42} C_VEL
LIN {X 0,Y 288.574,Z 817.137,A -85,B 0,C 180,E1 10244.938,E2 10244.938} C_VEL
LIN {X 0,Y 289.223,Z 817.082,A -85,B 0,C 180,E1 10244.459,E2 10244.459} C_VEL
LIN {X 0,Y 292.78,Z 823.194,A -85,B 0,C 180,E1 10241.585,E2 10241.585} C_VEL
LIN {X 0,Y 298.072,Z 833.04,A -85,B 0,C 180,E1 10238.036,E2 10238.036} C_VEL
LIN {X 0,Y 303.532,Z 843.918,A -85,B 0,C 180,E1 10234.947,E2 10234.947} C_VEL
LIN {X 0,Y 305.729,Z 848.909,A -85,B 0,C 180,E1 10233.798,E2 10233.798} C_VEL
LIN {X 0,Y 289.157,Z 1052.175,A -85,B 0,C 180,E1 10229.435,E2 10229.435} C_VEL
LIN {X 0,Y 286.321,Z 1072.712,A -85,B 0,C 180,E1 10228.715,E2 10228.715} C_VEL
LIN {X 0,Y 282.307,Z 1092.824,A -85,B 0,C 180,E1 10227.724,E2 10227.724} C_VEL
LIN {X 0,Y 277.54,Z 1111.243,A -85,B 0,C 180,E1 10226.528,E2 10226.528} C_VEL
LIN {X 0,Y 271.611,Z 1129.834,A -85,B 0,C 180,E1 10224.99,E2 10224.99} C_VEL
LIN {X 0,Y 264.757,Z 1147.784,A -85,B 0,C 180,E1 10223.096,E2 10223.096} C_VEL
LIN {X 0,Y 257.538,Z 1164.102,A -85,B 0,C 180,E1 10220.937,E2 10220.937} C_VEL
LIN {X 0,Y 249.712,Z 1179.819,A -85,B 0,C 180,E1 10218.342,E2 10218.342} C_VEL
LIN {X 0,Y 241.183,Z 1195.21,A -85,B 0,C 180,E1 10215.144,E2 10215.144} C_VEL
LIN {X 0,Y 233.178,Z 1208.478,A -85,B 0,C 180,E1 10211.653,E2 10211.653} C_VEL
LIN {X 0,Y 225.559,Z 1220.331,A -85,B 0,C 180,E1 10207.713,E2 10207.713} C_VEL
LIN {X 0,Y 218.578,Z 1230.76,A -85,B 0,C 180,E1 10203.292,E2 10203.292} C_VEL
LIN {X 0,Y 212.197,Z 1240.116,A -85,B 0,C 180,E1 10198.11,E2 10198.11} C_VEL
LIN {X 0,Y 207.317,Z 1247.434,A -85,B 0,C 180,E1 10192.694,E2 10192.694} C_VEL
LIN {X 0,Y 203.919,Z 1252.929,A -85,B 0,C 180,E1 10187.108,E2 10187.108} C_VEL
LIN {X 0,Y 201.815,Z 1256.875,A -85,B 0,C 180,E1 10181.196,E2 10181.196} C_VEL
LIN {X 0,Y 200.893,Z 1259.092,A -85,B 0,C 180,E1 10175.425,E2 10175.425} C_VEL
LIN {X 0,Y 200.687,Z 1259.82,A -85,B 0,C 180,E1 10169.999,E2 10169.999} C_VEL
LIN {X 0,Y 200.891,Z 1259.112,A -85,B 0,C 180,E1 10164.523,E2 10164.523} C_VEL
LIN {X 0,Y 201.787,Z 1256.968,A -85,B 0,C 180,E1 10158.844,E2 10158.844} C_VEL
LIN {X 0,Y 203.795,Z 1253.202,A -85,B 0,C 180,E1 10153.081,E2 10153.081} C_VEL
LIN {X 0,Y 207.061,Z 1247.916,A -85,B 0,C 180,E1 10147.574,E2 10147.574} C_VEL
LIN {X 0,Y 211.845,Z 1240.706,A -85,B 0,C 180,E1 10142.142,E2 10142.142} C_VEL
LIN {X 0,Y 217.887,Z 1231.824,A -85,B 0,C 180,E1 10137.116,E2 10137.116} C_VEL
LIN {X 0,Y 224.624,Z 1221.82,A -85,B 0,C 180,E1 10132.743,E2 10132.743} C_VEL
LIN {X 0,Y 232.124,Z 1210.287,A -85,B 0,C 180,E1 10128.772,E2 10128.772} C_VEL
LIN {X 0,Y 240.027,Z 1197.388,A -85,B 0,C 180,E1 10125.251,E2 10125.251} C_VEL
LIN {X 0,Y 248.128,Z 1183.078,A -85,B 0,C 180,E1 10122.144,E2 10122.144} C_VEL
LIN {X 0,Y 256.231,Z 1167.219,A -85,B 0,C 180,E1 10119.408,E2 10119.408} C_VEL
LIN {X 0,Y 263.883,Z 1150.191,A -85,B 0,C 180,E1 10117.08,E2 10117.08} C_VEL
LIN {X 0,Y 266.261,Z 1144.17,A -85,B 0,C 180,E1 10116.36,E2 10116.36} C_VEL
LIN {X 0,Y 263.084,Z 1146.228,A -85,B 0,C 180,E1 10115.823,E2 10115.823} C_VEL
LIN {X 0,Y 255.502,Z 1151.436,A -85,B 0,C 180,E1 10114.572,E2 10114.572} C_VEL
LIN {X 0,Y 248.687,Z 1155.252,A -85,B 0,C 180,E1 10113.148,E2 10113.148} C_VEL
LIN {X 0,Y 241.904,Z 1159.294,A -85,B 0,C 180,E1 10111.664,E2 10111.664} C_VEL
LIN {X 0,Y 237.928,Z 1161.209,A -85,B 0,C 180,E1 10110.564,E2 10110.564} C_VEL
LIN {X 0,Y 231.659,Z 1164.633,A -85,B 0,C 180,E1 10108.908,E2 10108.908} C_VEL
LIN {X 0,Y 228.075,Z 1166.164,A -85,B 0,C 180,E1 10107.679,E2 10107.679} C_VEL
LIN {X 0,Y 223.115,Z 1168.776,A -85,B 0,C 180,E1 10106.052,E2 10106.052} C_VEL
LIN {X 0,Y 220.022,Z 1169.984,A -85,B 0,C 180,E1 10104.714,E2 10104.714} C_VEL
LIN {X 0,Y 216.082,Z 1172.096,A -85,B 0,C 180,E1 10103.161,E2 10103.161} C_VEL
LIN {X 0,Y 213.54,Z 1172.902,A -85,B 0,C 180,E1 10101.71,E2 10101.71} C_VEL
LIN {X 0,Y 209.95,Z 1174.88,A -85,B 0,C 180,E1 10100.054,E2 10100.054} C_VEL
LIN {X 0,Y 207.948,Z 1175.356,A -85,B 0,C 180,E1 10098.503,E2 10098.503} C_VEL
LIN {X 0,Y 207.746,Z 1176.232,A -85,B 0,C 180,E1 10098.166,E2 10098.166} C_VEL
LIN {X 0,Y 205.82,Z 1180.721,A -85,B 0,C 180,E1 10096.483,E2 10096.483} C_VEL
LIN {X 0,Y 198.046,Z 1191.175,A -85,B 0,C 180,E1 10092.126,E2 10092.126} C_VEL
LIN {X 0,Y 196.531,Z 1194.842,A -85,B 0,C 180,E1 10090.183,E2 10090.183} C_VEL
LIN {X 0,Y 195.827,Z 1202.941,A -85,B 0,C 180,E1 10084.98,E2 10084.98} C_VEL
LIN {X 0,Y 196.069,Z 1209.146,A -85,B 0,C 180,E1 10079.708,E2 10079.708} C_VEL
LIN {X 0,Y 197.38,Z 1213.953,A -85,B 0,C 180,E1 10074.186,E2 10074.186} C_VEL
LIN {X 0,Y 200.117,Z 1217.072,A -85,B 0,C 180,E1 10068.472,E2 10068.472} C_VEL
LIN {X 0,Y 204.449,Z 1218.424,A -85,B 0,C 180,E1 10062.937,E2 10062.937} C_VEL
LIN {X 0,Y 210.847,Z 1218.048,A -85,B 0,C 180,E1 10057.412,E2 10057.412} C_VEL
LIN {X 0,Y 220.08,Z 1215.613,A -85,B 0,C 180,E1 10051.805,E2 10051.805} C_VEL
LIN {X 0,Y 231.555,Z 1211.208,A -85,B 0,C 180,E1 10046.744,E2 10046.744} C_VEL
LIN {X 0,Y 242.226,Z 1206.499,A -85,B 0,C 180,E1 10043.118,E2 10043.118} C_VEL
LIN {X 0,Y 229.571,Z 1216.77,A -85,B 0,C 180,E1 10039.275,E2 10039.275} C_VEL
LIN {X 0,Y 221.862,Z 1230.435,A -85,B 0,C 180,E1 10035.772,E2 10035.772} C_VEL
LIN {X 0,Y 214.142,Z 1243.51,A -85,B 0,C 180,E1 10031.532,E2 10031.532} C_VEL
LIN {X 0,Y 207.198,Z 1255.134,A -85,B 0,C 180,E1 10026.755,E2 10026.755} C_VEL
LIN {X 0,Y 201.36,Z 1265.276,A -85,B 0,C 180,E1 10021.426,E2 10021.426} C_VEL
LIN {X 0,Y 196.91,Z 1273.871,A -85,B 0,C 180,E1 10015.571,E2 10015.571} C_VEL
LIN {X 0,Y 194.11,Z 1280.535,A -85,B 0,C 180,E1 10009.563,E2 10009.563} C_VEL
LIN {X 0,Y 192.785,Z 1285.399,A -85,B 0,C 180,E1 10003.498,E2 10003.498} C_VEL
LIN {X 0,Y 192.55,Z 1288.187,A -85,B 0,C 180,E1 9998.061,E2 9998.061} C_VEL
LIN {X 0,Y 192.72,Z 1289.607,A -85,B 0,C 180,E1 9992.975,E2 9992.975} C_VEL
LIN {X 0,Y 192.762,Z 1289.736,A -85,B 0,C 180,E1 9988.515,E2 9988.515} C_VEL
LIN {X 0,Y 192.587,Z 1288.839,A -85,B 0,C 180,E1 9983.742,E2 9983.742} C_VEL
LIN {X 0,Y 192.579,Z 1286.423,A -85,B 0,C 180,E1 9978.319,E2 9978.319} C_VEL
LIN {X 0,Y 193.383,Z 1282.404,A -85,B 0,C 180,E1 9972.551,E2 9972.551} C_VEL
LIN {X 0,Y 195.573,Z 1276.419,A -85,B 0,C 180,E1 9966.5,E2 9966.5} C_VEL
LIN {X 0,Y 199.386,Z 1268.484,A -85,B 0,C 180,E1 9960.566,E2 9960.566} C_VEL
LIN {X 0,Y 204.6,Z 1259.033,A -85,B 0,C 180,E1 9955.128,E2 9955.128} C_VEL
LIN {X 0,Y 211.133,Z 1247.86,A -85,B 0,C 180,E1 9950.1,E2 9950.1} C_VEL
LIN {X 0,Y 218.617,Z 1235.13,A -85,B 0,C 180,E1 9945.595,E2 9945.595} C_VEL
LIN {X 0,Y 226.737,Z 1220.923,A -85,B 0,C 180,E1 9941.632,E2 9941.632} C_VEL
LIN {X 0,Y 234.976,Z 1205.695,A -85,B 0,C 180,E1 9938.274,E2 9938.274} C_VEL
LIN {X 0,Y 242.988,Z 1189.593,A -85,B 0,C 180,E1 9935.441,E2 9935.441} C_VEL
LIN {X 0,Y 250.569,Z 1172.615,A -85,B 0,C 180,E1 9933.075,E2 9933.075} C_VEL
LIN {X 0,Y 257.665,Z 1154.489,A -85,B 0,C 180,E1 9931.07,E2 9931.07} C_VEL
LIN {X 0,Y 264.004,Z 1135.536,A -85,B 0,C 180,E1 9929.419,E2 9929.419} C_VEL
LIN {X 0,Y 269.621,Z 1115.042,A -85,B 0,C 180,E1 9928.045,E2 9928.045} C_VEL
LIN {X 0,Y 274.047,Z 1094.235,A -85,B 0,C 180,E1 9927.028,E2 9927.028} C_VEL
LIN {X 0,Y 277.098,Z 1073.895,A -85,B 0,C 180,E1 9926.325,E2 9926.325} C_VEL
LIN {X 0,Y 281.182,Z 1027.521,A -85,B 0,C 180,E1 9925.263,E2 9925.263} C_VEL
LIN {X 0,Y 284.147,Z 1001.042,A -85,B 0,C 180,E1 9924.995,E2 9924.995} C_VEL
LIN {X 0,Y 287.868,Z 974.576,A -85,B 0,C 180,E1 9925.048,E2 9925.048} C_VEL
LIN {X 0,Y 288.196,Z 972.014,A -85,B 0,C 180,E1 9925.04,E2 9925.04} C_VEL
LIN {X 0,Y 284.365,Z 949.717,A -85,B 0,C 180,E1 9921.964,E2 9921.964} C_VEL
LIN {X 0,Y 283.523,Z 940.155,A -85,B 0,C 180,E1 9920.768,E2 9920.768} C_VEL
LIN {X 0,Y 285.71,Z 915.101,A -85,B 0,C 180,E1 9917.184,E2 9917.184} C_VEL
LIN {X 0,Y 290.283,Z 889.796,A -85,B 0,C 180,E1 9913.952,E2 9913.952} C_VEL
LIN {X 0,Y 291.857,Z 882.829,A -85,B 0,C 180,E1 9913.118,E2 9913.118} C_VEL
LIN {X 0,Y 284.55,Z 867.546,A -85,B 0,C 180,E1 9908.486,E2 9908.486} C_VEL
LIN {X 0,Y 277.774,Z 854.025,A -85,B 0,C 180,E1 9903.921,E2 9903.921} C_VEL
LIN {X 0,Y 275.521,Z 849.444,A -85,B 0,C 180,E1 9902.183,E2 9902.183} C_VEL
LIN {X 0,Y 275.867,Z 844.315,A -85,B 0,C 180,E1 9899.48,E2 9899.48} C_VEL
LIN {X 0,Y 277.3,Z 837.924,A -85,B 0,C 180,E1 9895.657,E2 9895.657} C_VEL
LIN {X 0,Y 278.694,Z 834.432,A -85,B 0,C 180,E1 9893.407,E2 9893.407} C_VEL
LIN {X 0,Y 280.56,Z 831.166,A -85,B 0,C 180,E1 9891.081,E2 9891.081} C_VEL
LIN {X 0,Y 282.606,Z 828.658,A -85,B 0,C 180,E1 9888.985,E2 9888.985} C_VEL
LIN {X 0,Y 287.895,Z 825.018,A -85,B 0,C 180,E1 9884.695,E2 9884.695} C_VEL
LIN {X 0,Y 291.249,Z 831.072,A -85,B 0,C 180,E1 9881.899,E2 9881.899} C_VEL
LIN {X 0,Y 295.91,Z 840.078,A -85,B 0,C 180,E1 9878.649,E2 9878.649} C_VEL
LIN {X 0,Y 301.015,Z 850.629,A -85,B 0,C 180,E1 9875.624,E2 9875.624} C_VEL
LIN {X 0,Y 301.973,Z 853.049,A -85,B 0,C 180,E1 9875.081,E2 9875.081} C_VEL
LIN {X 0,Y 285.167,Z 1052.829,A -85,B 0,C 180,E1 9870.812,E2 9870.812} C_VEL
LIN {X 0,Y 282.246,Z 1073.344,A -85,B 0,C 180,E1 9870.097,E2 9870.097} C_VEL
LIN {X 0,Y 278.125,Z 1093.402,A -85,B 0,C 180,E1 9869.114,E2 9869.114} C_VEL
LIN {X 0,Y 273.214,Z 1111.832,A -85,B 0,C 180,E1 9867.926,E2 9867.926} C_VEL
LIN {X 0,Y 267.102,Z 1130.429,A -85,B 0,C 180,E1 9866.395,E2 9866.395} C_VEL
LIN {X 0,Y 259.994,Z 1148.459,A -85,B 0,C 180,E1 9864.5,E2 9864.5} C_VEL
LIN {X 0,Y 252.555,Z 1164.707,A -85,B 0,C 180,E1 9862.352,E2 9862.352} C_VEL
LIN {X 0,Y 244.35,Z 1180.595,A -85,B 0,C 180,E1 9859.72,E2 9859.72} C_VEL
LIN {X 0,Y 235.571,Z 1195.821,A -85,B 0,C 180,E1 9856.533,E2 9856.533} C_VEL
LIN {X 0,Y 227.21,Z 1209.092,A -85,B 0,C 180,E1 9853.006,E2 9853.006} C_VEL
LIN {X 0,Y 219.222,Z 1220.946,A -85,B 0,C 180,E1 9849.005,E2 9849.005} C_VEL
LIN {X 0,Y 211.865,Z 1231.376,A -85,B 0,C 180,E1 9844.492,E2 9844.492} C_VEL
LIN {X 0,Y 205.1,Z 1240.733,A -85,B 0,C 180,E1 9839.175,E2 9839.175} C_VEL
LIN {X 0,Y 199.888,Z 1248.051,A -85,B 0,C 180,E1 9833.587,E2 9833.587} C_VEL
LIN {X 0,Y 196.228,Z 1253.545,A -85,B 0,C 180,E1 9827.8,E2 9827.8} C_VEL
LIN {X 0,Y 194.013,Z 1257.368,A -85,B 0,C 180,E1 9821.895,E2 9821.895} C_VEL
LIN {X 0,Y 192.966,Z 1259.64,A -85,B 0,C 180,E1 9815.947,E2 9815.947} C_VEL
LIN {X 0,Y 192.704,Z 1260.387,A -85,B 0,C 180,E1 9810.593,E2 9810.593} C_VEL
LIN {X 0,Y 192.878,Z 1259.857,A -85,B 0,C 180,E1 9804.943,E2 9804.943} C_VEL
LIN {X 0,Y 193.77,Z 1257.885,A -85,B 0,C 180,E1 9798.992,E2 9798.992} C_VEL
LIN {X 0,Y 195.784,Z 1254.37,A -85,B 0,C 180,E1 9793.075,E2 9793.075} C_VEL
LIN {X 0,Y 199.4,Z 1248.842,A -85,B 0,C 180,E1 9786.975,E2 9786.975} C_VEL
LIN {X 0,Y 204.432,Z 1241.706,A -85,B 0,C 180,E1 9781.359,E2 9781.359} C_VEL
LIN {X 0,Y 210.656,Z 1233.085,A -85,B 0,C 180,E1 9776.265,E2 9776.265} C_VEL
LIN {X 0,Y 217.812,Z 1223.045,A -85,B 0,C 180,E1 9771.704,E2 9771.704} C_VEL
LIN {X 0,Y 226.115,Z 1210.895,A -85,B 0,C 180,E1 9767.424,E2 9767.424} C_VEL
LIN {X 0,Y 234.371,Z 1197.994,A -85,B 0,C 180,E1 9763.863,E2 9763.863} C_VEL
LIN {X 0,Y 242.803,Z 1183.68,A -85,B 0,C 180,E1 9760.736,E2 9760.736} C_VEL
LIN {X 0,Y 251.207,Z 1167.817,A -85,B 0,C 180,E1 9757.992,E2 9757.992} C_VEL
LIN {X 0,Y 256.972,Z 1155.533,A -85,B 0,C 180,E1 9756.259,E2 9756.259} C_VEL
LIN {X 0,Y 249.083,Z 1159.948,A -85,B 0,C 180,E1 9754.752,E2 9754.752} C_VEL
LIN {X 0,Y 240.406,Z 1164.814,A -85,B 0,C 180,E1 9753.014,E2 9753.014} C_VEL
LIN {X 0,Y 234.763,Z 1167.543,A -85,B 0,C 180,E1 9751.59,E2 9751.59} C_VEL
LIN {X 0,Y 228.243,Z 1170.869,A -85,B 0,C 180,E1 9749.844,E2 9749.844} C_VEL
LIN {X 0,Y 224.737,Z 1172.355,A -85,B 0,C 180,E1 9748.718,E2 9748.718} C_VEL
LIN {X 0,Y 219.088,Z 1175.006,A -85,B 0,C 180,E1 9746.861,E2 9746.861} C_VEL
LIN {X 0,Y 216.366,Z 1176.059,A -85,B 0,C 180,E1 9745.747,E2 9745.747} C_VEL
LIN {X 0,Y 211.824,Z 1178.223,A -85,B 0,C 180,E1 9743.951,E2 9743.951} C_VEL
LIN {X 0,Y 209.015,Z 1179.251,A -85,B 0,C 180,E1 9742.501,E2 9742.501} C_VEL
LIN {X 0,Y 205.091,Z 1181.129,A -85,B 0,C 180,E1 9740.55,E2 9740.55} C_VEL
LIN {X 0,Y 203.268,Z 1181.657,A -85,B 0,C 180,E1 9739.243,E2 9739.243} C_VEL
LIN {X 0,Y 199.794,Z 1183.486,A -85,B 0,C 180,E1 9737.174,E2 9737.174} C_VEL
LIN {X 0,Y 198.42,Z 1183.79,A -85,B 0,C 180,E1 9735.743,E2 9735.743} C_VEL
LIN {X 0,Y 196.692,Z 1193.705,A -85,B 0,C 180,E1 9730.842,E2 9730.842} C_VEL
LIN {X 0,Y 196.531,Z 1194.842,A -85,B 0,C 180,E1 9730.183,E2 9730.183} C_VEL
LIN {X 0,Y 195.162,Z 1198.3,A -85,B 0,C 180,E1 9728.188,E2 9728.188} C_VEL
LIN {X 0,Y 190.063,Z 1204.601,A -85,B 0,C 180,E1 9724.193,E2 9724.193} C_VEL
LIN {X 0,Y 188.126,Z 1207.818,A -85,B 0,C 180,E1 9721.729,E2 9721.729} C_VEL
LIN {X 0,Y 187.993,Z 1208.895,A -85,B 0,C 180,E1 9720.767,E2 9720.767} C_VEL
LIN {X 0,Y 189.108,Z 1214.205,A -85,B 0,C 180,E1 9715.148,E2 9715.148} C_VEL
LIN {X 0,Y 191.877,Z 1218.192,A -85,B 0,C 180,E1 9708.884,E2 9708.884} C_VEL
LIN {X 0,Y 196.218,Z 1220.146,A -85,B 0,C 180,E1 9703.116,E2 9703.116} C_VEL
LIN {X 0,Y 202.699,Z 1220.449,A -85,B 0,C 180,E1 9697.372,E2 9697.372} C_VEL
LIN {X 0,Y 211.647,Z 1218.911,A -85,B 0,C 180,E1 9691.809,E2 9691.809} C_VEL
LIN {X 0,Y 223.831,Z 1215.249,A -85,B 0,C 180,E1 9686.365,E2 9686.365} C_VEL
LIN {X 0,Y 232.663,Z 1212.024,A -85,B 0,C 180,E1 9683.321,E2 9683.321} C_VEL
LIN {X 0,Y 221.734,Z 1220.527,A -85,B 0,C 180,E1 9679.848,E2 9679.848} C_VEL
LIN {X 0,Y 213.109,Z 1234.642,A -85,B 0,C 180,E1 9675.878,E2 9675.878} C_VEL
LIN {X 0,Y 204.923,Z 1247.64,A -85,B 0,C 180,E1 9671.201,E2 9671.201} C_VEL
LIN {X 0,Y 197.958,Z 1258.698,A -85,B 0,C 180,E1 9666.087,E2 9666.087} C_VEL
LIN {X 0,Y 192.396,Z 1267.916,A -85,B 0,C 180,E1 9660.618,E2 9660.618} C_VEL
LIN {X 0,Y 188.16,Z 1275.833,A -85,B 0,C 180,E1 9654.488,E2 9654.488} C_VEL
LIN {X 0,Y 185.651,Z 1281.813,A -85,B 0,C 180,E1 9648.203,E2 9648.203} C_VEL
LIN {X 0,Y 184.668,Z 1285.826,A -85,B 0,C 180,E1 9642.192,E2 9642.192} C_VEL
LIN {X 0,Y 184.624,Z 1288.312,A -85,B 0,C 180,E1 9636.219,E2 9636.219} C_VEL
LIN {X 0,Y 184.785,Z 1289.129,A -85,B 0,C 180,E1 9631.552,E2 9631.552} C_VEL
LIN {X 0,Y 184.732,Z 1288.994,A -85,B 0,C 180,E1 9626.899,E2 9626.899} C_VEL
LIN {X 0,Y 184.536,Z 1287.555,A -85,B 0,C 180,E1 9621.589,E2 9621.589} C_VEL
LIN {X 0,Y 184.785,Z 1284.75,A -85,B 0,C 180,E1 9615.909,E2 9615.909} C_VEL
LIN {X 0,Y 186.23,Z 1279.87,A -85,B 0,C 180,E1 9609.577,E2 9609.577} C_VEL
LIN {X 0,Y 189.273,Z 1273.185,A -85,B 0,C 180,E1 9603.321,E2 9603.321} C_VEL
LIN {X 0,Y 194.056,Z 1264.565,A -85,B 0,C 180,E1 9597.25,E2 9597.25} C_VEL
LIN {X 0,Y 200.26,Z 1254.396,A -85,B 0,C 180,E1 9591.751,E2 9591.751} C_VEL
LIN {X 0,Y 207.599,Z 1242.746,A -85,B 0,C 180,E1 9586.852,E2 9586.852} C_VEL
LIN {X 0,Y 215.583,Z 1229.935,A -85,B 0,C 180,E1 9582.62,E2 9582.62} C_VEL
LIN {X 0,Y 224.377,Z 1215.06,A -85,B 0,C 180,E1 9578.758,E2 9578.758} C_VEL
LIN {X 0,Y 233.258,Z 1198.852,A -85,B 0,C 180,E1 9575.471,E2 9575.471} C_VEL
LIN {X 0,Y 241.83,Z 1181.525,A -85,B 0,C 180,E1 9572.716,E2 9572.716} C_VEL
LIN {X 0,Y 249.552,Z 1163.943,A -85,B 0,C 180,E1 9570.526,E2 9570.526} C_VEL
LIN {X 0,Y 256.518,Z 1145.623,A -85,B 0,C 180,E1 9568.719,E2 9568.719} C_VEL
LIN {X 0,Y 262.996,Z 1125.339,A -85,B 0,C 180,E1 9567.177,E2 9567.177} C_VEL
LIN {X 0,Y 267.984,Z 1105.92,A -85,B 0,C 180,E1 9566.061,E2 9566.061} C_VEL
LIN {X 0,Y 271.846,Z 1086.018,A -85,B 0,C 180,E1 9565.207,E2 9565.207} C_VEL
LIN {X 0,Y 274.616,Z 1064.386,A -85,B 0,C 180,E1 9564.591,E2 9564.591} C_VEL
LIN {X 0,Y 277.798,Z 1027.604,A -85,B 0,C 180,E1 9563.777,E2 9563.777} C_VEL
LIN {X 0,Y 280.817,Z 1000.94,A -85,B 0,C 180,E1 9563.519,E2 9563.519} C_VEL
LIN {X 0,Y 284.488,Z 974.013,A -85,B 0,C 180,E1 9563.546,E2 9563.546} C_VEL
LIN {X 0,Y 281.398,Z 954.172,A -85,B 0,C 180,E1 9560.758,E2 9560.758} C_VEL
LIN {X 0,Y 279.194,Z 928.504,A -85,B 0,C 180,E1 9557.574,E2 9557.574} C_VEL
LIN {X 0,Y 279.122,Z 921.18,A -85,B 0,C 180,E1 9556.76,E2 9556.76} C_VEL
LIN {X 0,Y 283.65,Z 895.488,A -85,B 0,C 180,E1 9553.376,E2 9553.376} C_VEL
LIN {X 0,Y 285.651,Z 886.859,A -85,B 0,C 180,E1 9552.328,E2 9552.328} C_VEL
LIN {X 0,Y 278.399,Z 871.685,A -85,B 0,C 180,E1 9547.636,E2 9547.636} C_VEL
LIN {X 0,Y 274.683,Z 864.007,A -85,B 0,C 180,E1 9545.011,E2 9545.011} C_VEL
LIN {X 0,Y 274.54,Z 855.748,A -85,B 0,C 180,E1 9540.939,E2 9540.939} C_VEL
LIN {X 0,Y 275.224,Z 850.366,A -85,B 0,C 180,E1 9538.022,E2 9538.022} C_VEL
LIN {X 0,Y 276.503,Z 845.611,A -85,B 0,C 180,E1 9535.229,E2 9535.229} C_VEL
LIN {X 0,Y 278.128,Z 841.859,A -85,B 0,C 180,E1 9532.771,E2 9532.771} C_VEL
LIN {X 0,Y 281.024,Z 837.314,A -85,B 0,C 180,E1 9529.545,E2 9529.545} C_VEL
LIN {X 0,Y 286.678,Z 833.125,A -85,B 0,C 180,E1 9524.836,E2 9524.836} C_VEL
LIN {X 0,Y 290.659,Z 840.73,A -85,B 0,C 180,E1 9521.498,E2 9521.498} C_VEL
LIN {X 0,Y 295.579,Z 850.886,A -85,B 0,C 180,E1 9518.102,E2 9518.102} C_VEL
LIN {X 0,Y 298.37,Z 857.222,A -85,B 0,C 180,E1 9516.396,E2 9516.396} C_VEL
LIN {X 0,Y 281.35,Z 1053.455,A -85,B 0,C 180,E1 9512.229,E2 9512.229} C_VEL
LIN {X 0,Y 278.337,Z 1074,A -85,B 0,C 180,E1 9511.517,E2 9511.517} C_VEL
LIN {X 0,Y 274.112,Z 1093.982,A -85,B 0,C 180,E1 9510.547,E2 9510.547} C_VEL
LIN {X 0,Y 269.056,Z 1112.42,A -85,B 0,C 180,E1 9509.368,E2 9509.368} C_VEL
LIN {X 0,Y 262.759,Z 1131.025,A -85,B 0,C 180,E1 9507.848,E2 9507.848} C_VEL
LIN {X 0,Y 255.397,Z 1149.126,A -85,B 0,C 180,E1 9505.955,E2 9505.955} C_VEL
LIN {X 0,Y 247.414,Z 1165.961,A -85,B 0,C 180,E1 9503.727,E2 9503.727} C_VEL
LIN {X 0,Y 238.96,Z 1181.682,A -85,B 0,C 180,E1 9501.1,E2 9501.1} C_VEL
LIN {X 0,Y 230.106,Z 1196.432,A -85,B 0,C 180,E1 9497.988,E2 9497.988} C_VEL
LIN {X 0,Y 221.376,Z 1209.706,A -85,B 0,C 180,E1 9494.43,E2 9494.43} C_VEL
LIN {X 0,Y 213.005,Z 1221.561,A -85,B 0,C 180,E1 9490.373,E2 9490.373} C_VEL
LIN {X 0,Y 205.251,Z 1231.993,A -85,B 0,C 180,E1 9485.771,E2 9485.771} C_VEL
LIN {X 0,Y 198.078,Z 1241.35,A -85,B 0,C 180,E1 9480.315,E2 9480.315} C_VEL
LIN {X 0,Y 192.51,Z 1248.668,A -85,B 0,C 180,E1 9474.549,E2 9474.549} C_VEL
LIN {X 0,Y 188.567,Z 1254.161,A -85,B 0,C 180,E1 9468.549,E2 9468.549} C_VEL
LIN {X 0,Y 186.163,Z 1257.981,A -85,B 0,C 180,E1 9462.404,E2 9462.404} C_VEL
LIN {X 0,Y 185.014,Z 1260.251,A -85,B 0,C 180,E1 9456.204,E2 9456.204} C_VEL
LIN {X 0,Y 184.727,Z 1260.996,A -85,B 0,C 180,E1 9450.619,E2 9450.619} C_VEL
LIN {X 0,Y 184.919,Z 1260.467,A -85,B 0,C 180,E1 9444.725,E2 9444.725} C_VEL
LIN {X 0,Y 185.896,Z 1258.497,A -85,B 0,C 180,E1 9438.52,E2 9438.52} C_VEL
LIN {X 0,Y 188.087,Z 1254.984,A -85,B 0,C 180,E1 9432.36,E2 9432.36} C_VEL
LIN {X 0,Y 191.99,Z 1249.457,A -85,B 0,C 180,E1 9426.031,E2 9426.031} C_VEL
LIN {X 0,Y 197.37,Z 1242.321,A -85,B 0,C 180,E1 9420.233,E2 9420.233} C_VEL
LIN {X 0,Y 203.977,Z 1233.698,A -85,B 0,C 180,E1 9415.003,E2 9415.003} C_VEL
LIN {X 0,Y 211.526,Z 1223.656,A -85,B 0,C 180,E1 9410.346,E2 9410.346} C_VEL
LIN {X 0,Y 220.237,Z 1211.504,A -85,B 0,C 180,E1 9406.003,E2 9406.003} C_VEL
LIN {X 0,Y 228.859,Z 1198.599,A -85,B 0,C 180,E1 9402.409,E2 9402.409} C_VEL
LIN {X 0,Y 237.632,Z 1184.281,A -85,B 0,C 180,E1 9399.266,E2 9399.266} C_VEL
LIN {X 0,Y 246.345,Z 1168.414,A -85,B 0,C 180,E1 9396.52,E2 9396.52} C_VEL
LIN {X 0,Y 247.654,Z 1165.509,A -85,B 0,C 180,E1 9396.047,E2 9396.047} C_VEL
LIN {X 0,Y 238.2,Z 1170.597,A -85,B 0,C 180,E1 9394.228,E2 9394.228} C_VEL
LIN {X 0,Y 232.343,Z 1173.271,A -85,B 0,C 180,E1 9392.836,E2 9392.836} C_VEL
LIN {X 0,Y 225.186,Z 1176.671,A -85,B 0,C 180,E1 9391.002,E2 9391.002} C_VEL
LIN {X 0,Y 221.195,Z 1178.383,A -85,B 0,C 180,E1 9389.784,E2 9389.784} C_VEL
LIN {X 0,Y 214.97,Z 1181.088,A -85,B 0,C 180,E1 9387.718,E2 9387.718} C_VEL
LIN {X 0,Y 212.019,Z 1182.288,A -85,B 0,C 180,E1 9386.617,E2 9386.617} C_VEL
LIN {X 0,Y 206.976,Z 1184.372,A -85,B 0,C 180,E1 9384.548,E2 9384.548} C_VEL
LIN {X 0,Y 205.025,Z 1185.057,A -85,B 0,C 180,E1 9383.572,E2 9383.572} C_VEL
LIN {X 0,Y 200.493,Z 1187.032,A -85,B 0,C 180,E1 9381.35,E2 9381.35} C_VEL
LIN {X 0,Y 198.483,Z 1187.693,A -85,B 0,C 180,E1 9380.033,E2 9380.033} C_VEL
LIN {X 0,Y 194.982,Z 1189.338,A -85,B 0,C 180,E1 9377.92,E2 9377.92} C_VEL
LIN {X 0,Y 193.027,Z 1190.008,A -85,B 0,C 180,E1 9376.244,E2 9376.244} C_VEL
LIN {X 0,Y 189.926,Z 1191.564,A -85,B 0,C 180,E1 9373.704,E2 9373.704} C_VEL
LIN {X 0,Y 189.161,Z 1191.737,A -85,B 0,C 180,E1 9372.517,E2 9372.517} C_VEL
LIN {X 0,Y 188.051,Z 1200.436,A -85,B 0,C 180,E1 9367.332,E2 9367.332} C_VEL
LIN {X 0,Y 187.911,Z 1207.718,A -85,B 0,C 180,E1 9361.83,E2 9361.83} C_VEL
LIN {X 0,Y 187.993,Z 1208.895,A -85,B 0,C 180,E1 9360.767,E2 9360.767} C_VEL
LIN {X 0,Y 187.291,Z 1211.361,A -85,B 0,C 180,E1 9358.53,E2 9358.53} C_VEL
LIN {X 0,Y 182.888,Z 1217.117,A -85,B 0,C 180,E1 9352.332,E2 9352.332} C_VEL
LIN {X 0,Y 183.097,Z 1218.515,A -85,B 0,C 180,E1 9350.288,E2 9350.288} C_VEL
LIN {X 0,Y 187.186,Z 1221.4,A -85,B 0,C 180,E1 9344.192,E2 9344.192} C_VEL
LIN {X 0,Y 193.802,Z 1222.634,A -85,B 0,C 180,E1 9337.876,E2 9337.876} C_VEL
LIN {X 0,Y 203.156,Z 1221.922,A -85,B 0,C 180,E1 9331.806,E2 9331.806} C_VEL
LIN {X 0,Y 215.482,Z 1219.19,A -85,B 0,C 180,E1 9326.165,E2 9326.165} C_VEL
LIN {X 0,Y 222.869,Z 1217.078,A -85,B 0,C 180,E1 9323.478,E2 9323.478} C_VEL
LIN {X 0,Y 214.457,Z 1223.119,A -85,B 0,C 180,E1 9320.71,E2 9320.71} C_VEL
LIN {X 0,Y 205.351,Z 1237.176,A -85,B 0,C 180,E1 9316.511,E2 9316.511} C_VEL
LIN {X 0,Y 196.972,Z 1249.636,A -85,B 0,C 180,E1 9311.682,E2 9311.682} C_VEL
LIN {X 0,Y 189.984,Z 1260,A -85,B 0,C 180,E1 9306.493,E2 9306.493} C_VEL
LIN {X 0,Y 184.203,Z 1268.986,A -85,B 0,C 180,E1 9300.681,E2 9300.681} C_VEL
LIN {X 0,Y 179.946,Z 1276.495,A -85,B 0,C 180,E1 9294.28,E2 9294.28} C_VEL
LIN {X 0,Y 177.54,Z 1282.05,A -85,B 0,C 180,E1 9287.871,E2 9287.871} C_VEL
LIN {X 0,Y 176.626,Z 1285.9,A -85,B 0,C 180,E1 9281.429,E2 9281.429} C_VEL
LIN {X 0,Y 176.667,Z 1287.929,A -85,B 0,C 180,E1 9275.523,E2 9275.523} C_VEL
LIN {X 0,Y 176.821,Z 1288.594,A -85,B 0,C 180,E1 9270.649,E2 9270.649} C_VEL
LIN {X 0,Y 176.709,Z 1288.221,A -85,B 0,C 180,E1 9265.783,E2 9265.783} C_VEL
LIN {X 0,Y 176.542,Z 1286.686,A -85,B 0,C 180,E1 9260.548,E2 9260.548} C_VEL
LIN {X 0,Y 177.015,Z 1283.468,A -85,B 0,C 180,E1 9254.27,E2 9254.27} C_VEL
LIN {X 0,Y 178.9,Z 1278.385,A -85,B 0,C 180,E1 9247.665,E2 9247.665} C_VEL
LIN {X 0,Y 182.536,Z 1271.427,A -85,B 0,C 180,E1 9241.184,E2 9241.184} C_VEL
LIN {X 0,Y 188.043,Z 1262.488,A -85,B 0,C 180,E1 9234.954,E2 9234.954} C_VEL
LIN {X 0,Y 194.569,Z 1252.568,A -85,B 0,C 180,E1 9229.649,E2 9229.649} C_VEL
LIN {X 0,Y 202.524,Z 1240.664,A -85,B 0,C 180,E1 9224.692,E2 9224.692} C_VEL
LIN {X 0,Y 211.275,Z 1227.278,A -85,B 0,C 180,E1 9220.367,E2 9220.367} C_VEL
LIN {X 0,Y 220.162,Z 1212.879,A -85,B 0,C 180,E1 9216.722,E2 9216.722} C_VEL
LIN {X 0,Y 229.202,Z 1197.034,A -85,B 0,C 180,E1 9213.573,E2 9213.573} C_VEL
LIN {X 0,Y 237.818,Z 1180.229,A -85,B 0,C 180,E1 9210.946,E2 9210.946} C_VEL
LIN {X 0,Y 245.843,Z 1162.511,A -85,B 0,C 180,E1 9208.785,E2 9208.785} C_VEL
LIN {X 0,Y 253.063,Z 1144.012,A -85,B 0,C 180,E1 9207.009,E2 9207.009} C_VEL
LIN {X 0,Y 259.428,Z 1124.609,A -85,B 0,C 180,E1 9205.572,E2 9205.572} C_VEL
LIN {X 0,Y 264.522,Z 1105.32,A -85,B 0,C 180,E1 9204.48,E2 9204.48} C_VEL
LIN {X 0,Y 268.559,Z 1085.157,A -85,B 0,C 180,E1 9203.64,E2 9203.64} C_VEL
LIN {X 0,Y 271.413,Z 1063.324,A -85,B 0,C 180,E1 9203.027,E2 9203.027} C_VEL
LIN {X 0,Y 274.618,Z 1027.57,A -85,B 0,C 180,E1 9202.254,E2 9202.254} C_VEL
LIN {X 0,Y 277.694,Z 1000.701,A -85,B 0,C 180,E1 9202.008,E2 9202.008} C_VEL
LIN {X 0,Y 281.005,Z 976.338,A -85,B 0,C 180,E1 9202.048,E2 9202.048} C_VEL
LIN {X 0,Y 278.479,Z 957.833,A -85,B 0,C 180,E1 9199.424,E2 9199.424} C_VEL
LIN {X 0,Y 276.655,Z 932.228,A -85,B 0,C 180,E1 9196.211,E2 9196.211} C_VEL
LIN {X 0,Y 276.209,Z 908.665,A -85,B 0,C 180,E1 9193.609,E2 9193.609} C_VEL
LIN {X 0,Y 276.56,Z 903.19,A -85,B 0,C 180,E1 9193.059,E2 9193.059} C_VEL
LIN {X 0,Y 279.317,Z 890.624,A -85,B 0,C 180,E1 9191.459,E2 9191.459} C_VEL
LIN {X 0,Y 274.53,Z 880.269,A -85,B 0,C 180,E1 9188.165,E2 9188.165} C_VEL
LIN {X 0,Y 273.428,Z 870.295,A -85,B 0,C 180,E1 9183.826,E2 9183.826} C_VEL
LIN {X 0,Y 273.581,Z 863.114,A -85,B 0,C 180,E1 9180.314,E2 9180.314} C_VEL
LIN {X 0,Y 274.418,Z 857.742,A -85,B 0,C 180,E1 9177.389,E2 9177.389} C_VEL
LIN {X 0,Y 275.841,Z 853.017,A -85,B 0,C 180,E1 9174.592,E2 9174.592} C_VEL
LIN {X 0,Y 277.848,Z 848.839,A -85,B 0,C 180,E1 9171.828,E2 9171.828} C_VEL
LIN {X 0,Y 280.657,Z 844.827,A -85,B 0,C 180,E1 9168.908,E2 9168.908} C_VEL
LIN {X 0,Y 285.572,Z 841.388,A -85,B 0,C 180,E1 9164.879,E2 9164.879} C_VEL
LIN {X 0,Y 289.613,Z 849.708,A -85,B 0,C 180,E1 9161.428,E2 9161.428} C_VEL
LIN {X 0,Y 294.356,Z 860.008,A -85,B 0,C 180,E1 9158.111,E2 9158.111} C_VEL
LIN {X 0,Y 294.901,Z 861.684,A -85,B 0,C 180,E1 9157.736,E2 9157.736} C_VEL
LIN {X 0,Y 277.709,Z 1054.081,A -85,B 0,C 180,E1 9153.684,E2 9153.684} C_VEL
LIN {X 0,Y 274.603,Z 1074.659,A -85,B 0,C 180,E1 9152.977,E2 9152.977} C_VEL
LIN {X 0,Y 270.111,Z 1095.21,A -85,B 0,C 180,E1 9151.985,E2 9151.985} C_VEL
LIN {X 0,Y 264.312,Z 1115.322,A -85,B 0,C 180,E1 9150.684,E2 9150.684} C_VEL
LIN {X 0,Y 257.877,Z 1133.38,A -85,B 0,C 180,E1 9149.182,E2 9149.182} C_VEL
LIN {X 0,Y 250.549,Z 1150.752,A -85,B 0,C 180,E1 9147.353,E2 9147.353} C_VEL
LIN {X 0,Y 242.093,Z 1167.867,A -85,B 0,C 180,E1 9145.064,E2 9145.064} C_VEL
LIN {X 0,Y 233.365,Z 1183.37,A -85,B 0,C 180,E1 9142.43,E2 9142.43} C_VEL
LIN {X 0,Y 224.203,Z 1197.942,A -85,B 0,C 180,E1 9139.298,E2 9139.298} C_VEL
LIN {X 0,Y 215.144,Z 1211.065,A -85,B 0,C 180,E1 9135.698,E2 9135.698} C_VEL
LIN {X 0,Y 206.428,Z 1222.789,A -85,B 0,C 180,E1 9131.571,E2 9131.571} C_VEL
LIN {X 0,Y 198.325,Z 1233.116,A -85,B 0,C 180,E1 9126.864,E2 9126.864} C_VEL
LIN {X 0,Y 190.802,Z 1242.387,A -85,B 0,C 180,E1 9121.249,E2 9121.249} C_VEL
LIN {X 0,Y 184.692,Z 1249.948,A -85,B 0,C 180,E1 9114.976,E2 9114.976} C_VEL
LIN {X 0,Y 180.455,Z 1255.496,A -85,B 0,C 180,E1 9108.409,E2 9108.409} C_VEL
LIN {X 0,Y 178.055,Z 1259.042,A -85,B 0,C 180,E1 9101.99,E2 9101.99} C_VEL
LIN {X 0,Y 176.969,Z 1261.048,A -85,B 0,C 180,E1 9095.51,E2 9095.51} C_VEL
LIN {X 0,Y 176.751,Z 1261.636,A -85,B 0,C 180,E1 9089.674,E2 9089.674} C_VEL
LIN {X 0,Y 177.032,Z 1260.934,A -85,B 0,C 180,E1 9083.741,E2 9083.741} C_VEL
LIN {X 0,Y 178.209,Z 1258.811,A -85,B 0,C 180,E1 9077.359,E2 9077.359} C_VEL
LIN {X 0,Y 180.737,Z 1255.119,A -85,B 0,C 180,E1 9070.948,E2 9070.948} C_VEL
LIN {X 0,Y 184.883,Z 1249.76,A -85,B 0,C 180,E1 9064.706,E2 9064.706} C_VEL
LIN {X 0,Y 190.803,Z 1242.462,A -85,B 0,C 180,E1 9058.669,E2 9058.669} C_VEL
LIN {X 0,Y 197.819,Z 1233.817,A -85,B 0,C 180,E1 9053.385,E2 9053.385} C_VEL
LIN {X 0,Y 205.844,Z 1223.655,A -85,B 0,C 180,E1 9048.653,E2 9048.653} C_VEL
LIN {X 0,Y 214.502,Z 1212.113,A -85,B 0,C 180,E1 9044.505,E2 9044.505} C_VEL
LIN {X 0,Y 223.504,Z 1199.205,A -85,B 0,C 180,E1 9040.883,E2 9040.883} C_VEL
LIN {X 0,Y 232.625,Z 1184.882,A -85,B 0,C 180,E1 9037.733,E2 9037.733} C_VEL
LIN {X 0,Y 238.092,Z 1175.195,A -85,B 0,C 180,E1 9035.936,E2 9035.936} C_VEL
LIN {X 0,Y 228.918,Z 1179.375,A -85,B 0,C 180,E1 9033.913,E2 9033.913} C_VEL
LIN {X 0,Y 221.163,Z 1182.693,A -85,B 0,C 180,E1 9031.935,E2 9031.935} C_VEL
LIN {X 0,Y 211.847,Z 1186.558,A -85,B 0,C 180,E1 9029.087,E2 9029.087} C_VEL
LIN {X 0,Y 208.215,Z 1187.979,A -85,B 0,C 180,E1 9027.763,E2 9027.763} C_VEL
LIN {X 0,Y 203.019,Z 1190.048,A -85,B 0,C 180,E1 9025.684,E2 9025.684} C_VEL
LIN {X 0,Y 200.393,Z 1190.988,A -85,B 0,C 180,E1 9024.465,E2 9024.465} C_VEL
LIN {X 0,Y 195.367,Z 1192.926,A -85,B 0,C 180,E1 9021.939,E2 9021.939} C_VEL
LIN {X 0,Y 193.109,Z 1193.78,A -85,B 0,C 180,E1 9020.615,E2 9020.615} C_VEL
LIN {X 0,Y 189.366,Z 1195.26,A -85,B 0,C 180,E1 9018.152,E2 9018.152} C_VEL
LIN {X 0,Y 187.951,Z 1195.778,A -85,B 0,C 180,E1 9017.014,E2 9017.014} C_VEL
LIN {X 0,Y 184.768,Z 1197.231,A -85,B 0,C 180,E1 9014.415,E2 9014.415} C_VEL
LIN {X 0,Y 183.504,Z 1197.692,A -85,B 0,C 180,E1 9012.909,E2 9012.909} C_VEL
LIN {X 0,Y 180.971,Z 1199.118,A -85,B 0,C 180,E1 9010.184,E2 9010.184} C_VEL
LIN {X 0,Y 180.23,Z 1199.589,A -85,B 0,C 180,E1 9008.491,E2 9008.491} C_VEL
LIN {X 0,Y 179.879,Z 1206.877,A -85,B 0,C 180,E1 9003.187,E2 9003.187} C_VEL
LIN {X 0,Y 180.611,Z 1213.319,A -85,B 0,C 180,E1 8997.145,E2 8997.145} C_VEL
LIN {X 0,Y 182.654,Z 1217.958,A -85,B 0,C 180,E1 8991.184,E2 8991.184} C_VEL
LIN {X 0,Y 183.097,Z 1218.515,A -85,B 0,C 180,E1 8990.288,E2 8990.288} C_VEL
LIN {X 0,Y 183.469,Z 1220.046,A -85,B 0,C 180,E1 8987.91,E2 8987.91} C_VEL
LIN {X 0,Y 182.358,Z 1223.551,A -85,B 0,C 180,E1 8981.529,E2 8981.529} C_VEL
LIN {X 0,Y 183.782,Z 1224.244,A -85,B 0,C 180,E1 8979.328,E2 8979.328} C_VEL
LIN {X 0,Y 191.906,Z 1224.754,A -85,B 0,C 180,E1 8973.381,E2 8973.381} C_VEL
LIN {X 0,Y 203.167,Z 1223.522,A -85,B 0,C 180,E1 8967.56,E2 8967.56} C_VEL
LIN {X 0,Y 213.101,Z 1221.506,A -85,B 0,C 180,E1 8963.642,E2 8963.642} C_VEL
LIN {X 0,Y 207.516,Z 1225.117,A -85,B 0,C 180,E1 8961.756,E2 8961.756} C_VEL
LIN {X 0,Y 198.066,Z 1238.804,A -85,B 0,C 180,E1 8957.434,E2 8957.434} C_VEL
LIN {X 0,Y 189.911,Z 1250.261,A -85,B 0,C 180,E1 8952.78,E2 8952.78} C_VEL
LIN {X 0,Y 182.237,Z 1260.969,A -85,B 0,C 180,E1 8947.124,E2 8947.124} C_VEL
LIN {X 0,Y 176.01,Z 1270.057,A -85,B 0,C 180,E1 8940.749,E2 8940.749} C_VEL
LIN {X 0,Y 171.737,Z 1277.156,A -85,B 0,C 180,E1 8934.052,E2 8934.052} C_VEL
LIN {X 0,Y 169.434,Z 1282.205,A -85,B 0,C 180,E1 8927.517,E2 8927.517} C_VEL
LIN {X 0,Y 168.615,Z 1285.706,A -85,B 0,C 180,E1 8920.94,E2 8920.94} C_VEL
LIN {X 0,Y 168.699,Z 1287.468,A -85,B 0,C 180,E1 8915.102,E2 8915.102} C_VEL
LIN {X 0,Y 168.857,Z 1288.024,A -85,B 0,C 180,E1 8910.002,E2 8910.002} C_VEL
LIN {X 0,Y 168.68,Z 1287.426,A -85,B 0,C 180,E1 8904.756,E2 8904.756} C_VEL
LIN {X 0,Y 168.574,Z 1285.687,A -85,B 0,C 180,E1 8899.06,E2 8899.06} C_VEL
LIN {X 0,Y 169.345,Z 1282.171,A -85,B 0,C 180,E1 8892.477,E2 8892.477} C_VEL
LIN {X 0,Y 171.743,Z 1276.784,A -85,B 0,C 180,E1 8885.586,E2 8885.586} C_VEL
LIN {X 0,Y 175.817,Z 1269.936,A -85,B 0,C 180,E1 8879.172,E2 8879.172} C_VEL
LIN {X 0,Y 181.966,Z 1260.875,A -85,B 0,C 180,E1 8872.815,E2 8872.815} C_VEL
LIN {X 0,Y 189.597,Z 1250.146,A -85,B 0,C 180,E1 8867.136,E2 8867.136} C_VEL
LIN {X 0,Y 198.287,Z 1237.861,A -85,B 0,C 180,E1 8862.165,E2 8862.165} C_VEL
LIN {X 0,Y 207.111,Z 1224.909,A -85,B 0,C 180,E1 8858.105,E2 8858.105} C_VEL
LIN {X 0,Y 216.559,Z 1210.181,A -85,B 0,C 180,E1 8854.501,E2 8854.501} C_VEL
LIN {X 0,Y 226.078,Z 1193.939,A -85,B 0,C 180,E1 8851.401,E2 8851.401} C_VEL
LIN {X 0,Y 234.763,Z 1177.448,A -85,B 0,C 180,E1 8848.931,E2 8848.931} C_VEL
LIN {X 0,Y 243.115,Z 1159.423,A -85,B 0,C 180,E1 8846.82,E2 8846.82} C_VEL
LIN {X 0,Y 250.609,Z 1140.382,A -85,B 0,C 180,E1 8845.09,E2 8845.09} C_VEL
LIN {X 0,Y 256.747,Z 1121.586,A -85,B 0,C 180,E1 8843.773,E2 8843.773} C_VEL
LIN {X 0,Y 262.085,Z 1101.087,A -85,B 0,C 180,E1 8842.688,E2 8842.688} C_VEL
LIN {X 0,Y 266.156,Z 1079.987,A -85,B 0,C 180,E1 8841.912,E2 8841.912} C_VEL
LIN {X 0,Y 268.863,Z 1057.268,A -85,B 0,C 180,E1 8841.313,E2 8841.313} C_VEL
LIN {X 0,Y 271.746,Z 1026.458,A -85,B 0,C 180,E1 8840.679,E2 8840.679} C_VEL
LIN {X 0,Y 274.951,Z 999.054,A -85,B 0,C 180,E1 8840.463,E2 8840.463} C_VEL
LIN {X 0,Y 277.671,Z 978.508,A -85,B 0,C 180,E1 8840.476,E2 8840.476} C_VEL
LIN {X 0,Y 275.58,Z 959.775,A -85,B 0,C 180,E1 8837.839,E2 8837.839} C_VEL
LIN {X 0,Y 274.273,Z 935.838,A -85,B 0,C 180,E1 8834.811,E2 8834.811} C_VEL
LIN {X 0,Y 274.138,Z 912.077,A -85,B 0,C 180,E1 8832.164,E2 8832.164} C_VEL
LIN {X 0,Y 274.511,Z 895.462,A -85,B 0,C 180,E1 8830.445,E2 8830.445} C_VEL
LIN {X 0,Y 272.989,Z 886.373,A -85,B 0,C 180,E1 8826.997,E2 8826.997} C_VEL
LIN {X 0,Y 272.311,Z 877.344,A -85,B 0,C 180,E1 8823.051,E2 8823.051} C_VEL
LIN {X 0,Y 272.675,Z 870.311,A -85,B 0,C 180,E1 8819.579,E2 8819.579} C_VEL
LIN {X 0,Y 273.691,Z 864.944,A -85,B 0,C 180,E1 8816.649,E2 8816.649} C_VEL
LIN {X 0,Y 275.214,Z 860.414,A -85,B 0,C 180,E1 8813.952,E2 8813.952} C_VEL
LIN {X 0,Y 278.428,Z 854.58,A -85,B 0,C 180,E1 8810.074,E2 8810.074} C_VEL
LIN {X 0,Y 280.993,Z 851.787,A -85,B 0,C 180,E1 8807.672,E2 8807.672} C_VEL
LIN {X 0,Y 284.34,Z 849.638,A -85,B 0,C 180,E1 8805.021,E2 8805.021} C_VEL
LIN {X 0,Y 288.073,Z 857.625,A -85,B 0,C 180,E1 8801.745,E2 8801.745} C_VEL
LIN {X 0,Y 291.616,Z 865.93,A -85,B 0,C 180,E1 8799.112,E2 8799.112} C_VEL
LIN {X 0,Y 274.253,Z 1054.704,A -85,B 0,C 180,E1 8795.176,E2 8795.176} C_VEL
LIN {X 0,Y 271.072,Z 1075.208,A -85,B 0,C 180,E1 8794.481,E2 8794.481} C_VEL
LIN {X 0,Y 266.454,Z 1095.788,A -85,B 0,C 180,E1 8793.501,E2 8793.501} C_VEL
LIN {X 0,Y 260.864,Z 1114.81,A -85,B 0,C 180,E1 8792.297,E2 8792.297} C_VEL
LIN {X 0,Y 254.209,Z 1133.167,A -85,B 0,C 180,E1 8790.809,E2 8790.809} C_VEL
LIN {X 0,Y 246.319,Z 1151.353,A -85,B 0,C 180,E1 8788.922,E2 8788.922} C_VEL
LIN {X 0,Y 237.587,Z 1168.472,A -85,B 0,C 180,E1 8786.651,E2 8786.651} C_VEL
LIN {X 0,Y 228.552,Z 1183.978,A -85,B 0,C 180,E1 8784.028,E2 8784.028} C_VEL
LIN {X 0,Y 219.037,Z 1198.553,A -85,B 0,C 180,E1 8780.895,E2 8780.895} C_VEL
LIN {X 0,Y 209.588,Z 1211.678,A -85,B 0,C 180,E1 8777.277,E2 8777.277} C_VEL
LIN {X 0,Y 200.457,Z 1223.404,A -85,B 0,C 180,E1 8773.103,E2 8773.103} C_VEL
LIN {X 0,Y 191.916,Z 1233.733,A -85,B 0,C 180,E1 8768.312,E2 8768.312} C_VEL
LIN {X 0,Y 183.935,Z 1243.004,A -85,B 0,C 180,E1 8762.556,E2 8762.556} C_VEL
LIN {X 0,Y 177.4,Z 1250.565,A -85,B 0,C 180,E1 8756.078,E2 8756.078} C_VEL
LIN {X 0,Y 172.825,Z 1256.111,A -85,B 0,C 180,E1 8749.253,E2 8749.253} C_VEL
LIN {X 0,Y 170.211,Z 1259.655,A -85,B 0,C 180,E1 8742.552,E2 8742.552} C_VEL
LIN {X 0,Y 169.015,Z 1261.658,A -85,B 0,C 180,E1 8735.77,E2 8735.77} C_VEL
LIN {X 0,Y 168.774,Z 1262.245,A -85,B 0,C 180,E1 8729.659,E2 8729.659} C_VEL
LIN {X 0,Y 169.086,Z 1261.542,A -85,B 0,C 180,E1 8723.437,E2 8723.437} C_VEL
LIN {X 0,Y 170.378,Z 1259.423,A -85,B 0,C 180,E1 8716.768,E2 8716.768} C_VEL
LIN {X 0,Y 173.133,Z 1255.733,A -85,B 0,C 180,E1 8710.077,E2 8710.077} C_VEL
LIN {X 0,Y 177.738,Z 1250.212,A -85,B 0,C 180,E1 8703.439,E2 8703.439} C_VEL
LIN {X 0,Y 184.219,Z 1242.763,A -85,B 0,C 180,E1 8697.127,E2 8697.127} C_VEL
LIN {X 0,Y 192.269,Z 1233.44,A -85,B 0,C 180,E1 8691.387,E2 8691.387} C_VEL
LIN {X 0,Y 201.388,Z 1222.426,A -85,B 0,C 180,E1 8686.359,E2 8686.359} C_VEL
LIN {X 0,Y 210.622,Z 1210.484,A -85,B 0,C 180,E1 8682.22,E2 8682.22} C_VEL
LIN {X 0,Y 220.163,Z 1197.112,A -85,B 0,C 180,E1 8678.635,E2 8678.635} C_VEL
LIN {X 0,Y 228.878,Z 1183.583,A -85,B 0,C 180,E1 8675.753,E2 8675.753} C_VEL
LIN {X 0,Y 220.172,Z 1187.45,A -85,B 0,C 180,E1 8673.791,E2 8673.791} C_VEL
LIN {X 0,Y 213.064,Z 1190.214,A -85,B 0,C 180,E1 8671.853,E2 8671.853} C_VEL
LIN {X 0,Y 198.93,Z 1195.483,A -85,B 0,C 180,E1 8666.896,E2 8666.896} C_VEL
LIN {X 0,Y 195.052,Z 1196.909,A -85,B 0,C 180,E1 8665.181,E2 8665.181} C_VEL
LIN {X 0,Y 190.122,Z 1198.629,A -85,B 0,C 180,E1 8662.577,E2 8662.577} C_VEL
LIN {X 0,Y 184.665,Z 1200.719,A -85,B 0,C 180,E1 8659.287,E2 8659.287} C_VEL
LIN {X 0,Y 182.714,Z 1201.404,A -85,B 0,C 180,E1 8657.789,E2 8657.789} C_VEL
LIN {X 0,Y 179.224,Z 1202.838,A -85,B 0,C 180,E1 8654.871,E2 8654.871} C_VEL
LIN {X 0,Y 177.765,Z 1203.442,A -85,B 0,C 180,E1 8653.334,E2 8653.334} C_VEL
LIN {X 0,Y 175.112,Z 1204.769,A -85,B 0,C 180,E1 8650.196,E2 8650.196} C_VEL
LIN {X 0,Y 174.12,Z 1205.309,A -85,B 0,C 180,E1 8648.587,E2 8648.587} C_VEL
LIN {X 0,Y 172.145,Z 1206.759,A -85,B 0,C 180,E1 8644.999,E2 8644.999} C_VEL
LIN {X 0,Y 171.906,Z 1207.19,A -85,B 0,C 180,E1 8643.502,E2 8643.502} C_VEL
LIN {X 0,Y 172.526,Z 1213.55,A -85,B 0,C 180,E1 8637.676,E2 8637.676} C_VEL
LIN {X 0,Y 174.835,Z 1219.142,A -85,B 0,C 180,E1 8630.786,E2 8630.786} C_VEL
LIN {X 0,Y 178.879,Z 1222.606,A -85,B 0,C 180,E1 8624.438,E2 8624.438} C_VEL
LIN {X 0,Y 183.782,Z 1224.244,A -85,B 0,C 180,E1 8619.328,E2 8619.328} C_VEL
LIN {X 0,Y 185.687,Z 1224.991,A -85,B 0,C 180,E1 8616.824,E2 8616.824} C_VEL
LIN {X 0,Y 188.577,Z 1226.763,A -85,B 0,C 180,E1 8610.926,E2 8610.926} C_VEL
LIN {X 0,Y 191.598,Z 1226.784,A -85,B 0,C 180,E1 8608.782,E2 8608.782} C_VEL
LIN {X 0,Y 203.246,Z 1225.459,A -85,B 0,C 180,E1 8603.785,E2 8603.785} C_VEL
LIN {X 0,Y 200.652,Z 1227.088,A -85,B 0,C 180,E1 8602.873,E2 8602.873} C_VEL
LIN {X 0,Y 190.951,Z 1240.263,A -85,B 0,C 180,E1 8598.486,E2 8598.486} C_VEL
LIN {X 0,Y 181.996,Z 1252.009,A -85,B 0,C 180,E1 8593.373,E2 8593.373} C_VEL
LIN {X 0,Y 174.137,Z 1262.265,A -85,B 0,C 180,E1 8587.492,E2 8587.492} C_VEL
LIN {X 0,Y 167.917,Z 1270.813,A -85,B 0,C 180,E1 8580.971,E2 8580.971} C_VEL
LIN {X 0,Y 163.689,Z 1277.472,A -85,B 0,C 180,E1 8574.16,E2 8574.16} C_VEL
LIN {X 0,Y 161.293,Z 1282.474,A -85,B 0,C 180,E1 8566.941,E2 8566.941} C_VEL
LIN {X 0,Y 160.602,Z 1285.594,A -85,B 0,C 180,E1 8560.041,E2 8560.041} C_VEL
LIN {X 0,Y 160.765,Z 1287.137,A -85,B 0,C 180,E1 8553.924,E2 8553.924} C_VEL
LIN {X 0,Y 160.858,Z 1287.349,A -85,B 0,C 180,E1 8548.933,E2 8548.933} C_VEL
LIN {X 0,Y 160.663,Z 1286.692,A -85,B 0,C 180,E1 8543.929,E2 8543.929} C_VEL
LIN {X 0,Y 160.661,Z 1284.633,A -85,B 0,C 180,E1 8537.421,E2 8537.421} C_VEL
LIN {X 0,Y 161.813,Z 1280.87,A -85,B 0,C 180,E1 8530.51,E2 8530.51} C_VEL
LIN {X 0,Y 164.815,Z 1275.182,A -85,B 0,C 180,E1 8523.327,E2 8523.327} C_VEL
LIN {X 0,Y 169.846,Z 1267.644,A -85,B 0,C 180,E1 8516.404,E2 8516.404} C_VEL
LIN {X 0,Y 176.54,Z 1258.629,A -85,B 0,C 180,E1 8510.211,E2 8510.211} C_VEL
LIN {X 0,Y 184.514,Z 1248.241,A -85,B 0,C 180,E1 8504.778,E2 8504.778} C_VEL
LIN {X 0,Y 193.897,Z 1235.759,A -85,B 0,C 180,E1 8499.797,E2 8499.797} C_VEL
LIN {X 0,Y 203.932,Z 1221.679,A -85,B 0,C 180,E1 8495.526,E2 8495.526} C_VEL
LIN {X 0,Y 213.874,Z 1206.584,A -85,B 0,C 180,E1 8492.018,E2 8492.018} C_VEL
LIN {X 0,Y 223.277,Z 1190.844,A -85,B 0,C 180,E1 8489.167,E2 8489.167} C_VEL
LIN {X 0,Y 232.366,Z 1173.858,A -85,B 0,C 180,E1 8486.768,E2 8486.768} C_VEL
LIN {X 0,Y 240.613,Z 1156.221,A -85,B 0,C 180,E1 8484.815,E2 8484.815} C_VEL
LIN {X 0,Y 248.036,Z 1137.657,A -85,B 0,C 180,E1 8483.21,E2 8483.21} C_VEL
LIN {X 0,Y 254.732,Z 1117.246,A -85,B 0,C 180,E1 8481.863,E2 8481.863} C_VEL
LIN {X 0,Y 260.179,Z 1095.89,A -85,B 0,C 180,E1 8480.846,E2 8480.846} C_VEL
LIN {X 0,Y 264.015,Z 1074.532,A -85,B 0,C 180,E1 8480.128,E2 8480.128} C_VEL
LIN {X 0,Y 267.406,Z 1041.8,A -85,B 0,C 180,E1 8479.349,E2 8479.349} C_VEL
LIN {X 0,Y 270.631,Z 1011.688,A -85,B 0,C 180,E1 8478.933,E2 8478.933} C_VEL
LIN {X 0,Y 274.36,Z 983.013,A -85,B 0,C 180,E1 8478.934,E2 8478.934} C_VEL
LIN {X 0,Y 274.594,Z 980.885,A -85,B 0,C 180,E1 8478.909,E2 8478.909} C_VEL
LIN {X 0,Y 272.925,Z 962.081,A -85,B 0,C 180,E1 8476.275,E2 8476.275} C_VEL
LIN {X 0,Y 272.058,Z 939.563,A -85,B 0,C 180,E1 8473.401,E2 8473.401} C_VEL
LIN {X 0,Y 272.243,Z 915.513,A -85,B 0,C 180,E1 8470.701,E2 8470.701} C_VEL
LIN {X 0,Y 272.718,Z 901.076,A -85,B 0,C 180,E1 8469.176,E2 8469.176} C_VEL
LIN {X 0,Y 271.673,Z 893.391,A -85,B 0,C 180,E1 8466.232,E2 8466.232} C_VEL
LIN {X 0,Y 271.244,Z 884.599,A -85,B 0,C 180,E1 8462.376,E2 8462.376} C_VEL
LIN {X 0,Y 271.787,Z 877.679,A -85,B 0,C 180,E1 8458.946,E2 8458.946} C_VEL
LIN {X 0,Y 273.178,Z 871.591,A -85,B 0,C 180,E1 8455.591,E2 8455.591} C_VEL
LIN {X 0,Y 274.772,Z 867.495,A -85,B 0,C 180,E1 8453.103,E2 8453.103} C_VEL
LIN {X 0,Y 278.039,Z 862.035,A -85,B 0,C 180,E1 8449.432,E2 8449.432} C_VEL
LIN {X 0,Y 280.727,Z 859.301,A -85,B 0,C 180,E1 8447.033,E2 8447.033} C_VEL
LIN {X 0,Y 283.111,Z 857.89,A -85,B 0,C 180,E1 8445.164,E2 8445.164} C_VEL
LIN {X 0,Y 286.296,Z 865.084,A -85,B 0,C 180,E1 8442.259,E2 8442.259} C_VEL
LIN {X 0,Y 288.468,Z 870.555,A -85,B 0,C 180,E1 8440.51,E2 8440.51} C_VEL
LIN {X 0,Y 270.986,Z 1055.328,A -85,B 0,C 180,E1 8436.705,E2 8436.705} C_VEL
LIN {X 0,Y 267.718,Z 1075.836,A -85,B 0,C 180,E1 8436.019,E2 8436.019} C_VEL
LIN {X 0,Y 262.95,Z 1096.509,A -85,B 0,C 180,E1 8435.05,E2 8435.05} C_VEL
LIN {X 0,Y 256.864,Z 1116.499,A -85,B 0,C 180,E1 8433.794,E2 8433.794} C_VEL
LIN {X 0,Y 250.057,Z 1134.571,A -85,B 0,C 180,E1 8432.332,E2 8432.332} C_VEL
LIN {X 0,Y 242.28,Z 1151.953,A -85,B 0,C 180,E1 8430.545,E2 8430.545} C_VEL
LIN {X 0,Y 232.92,Z 1169.726,A -85,B 0,C 180,E1 8428.204,E2 8428.204} C_VEL
LIN {X 0,Y 223.251,Z 1185.667,A -85,B 0,C 180,E1 8425.492,E2 8425.492} C_VEL
LIN {X 0,Y 213.412,Z 1200.064,A -85,B 0,C 180,E1 8422.35,E2 8422.35} C_VEL
LIN {X 0,Y 203.612,Z 1213.038,A -85,B 0,C 180,E1 8418.703,E2 8418.703} C_VEL
LIN {X 0,Y 193.573,Z 1225.245,A -85,B 0,C 180,E1 8414.21,E2 8414.21} C_VEL
LIN {X 0,Y 184.648,Z 1235.407,A -85,B 0,C 180,E1 8409.254,E2 8409.254} C_VEL
LIN {X 0,Y 176.79,Z 1244.008,A -85,B 0,C 180,E1 8403.657,E2 8403.657} C_VEL
LIN {X 0,Y 170.179,Z 1251.182,A -85,B 0,C 180,E1 8397.274,E2 8397.274} C_VEL
LIN {X 0,Y 165.233,Z 1256.727,A -85,B 0,C 180,E1 8390.175,E2 8390.175} C_VEL
LIN {X 0,Y 162.384,Z 1260.268,A -85,B 0,C 180,E1 8383.167,E2 8383.167} C_VEL
LIN {X 0,Y 161.064,Z 1262.268,A -85,B 0,C 180,E1 8376.056,E2 8376.056} C_VEL
LIN {X 0,Y 160.797,Z 1262.854,A -85,B 0,C 180,E1 8369.642,E2 8369.642} C_VEL
LIN {X 0,Y 161.143,Z 1262.152,A -85,B 0,C 180,E1 8363.112,E2 8363.112} C_VEL
LIN {X 0,Y 162.561,Z 1260.036,A -85,B 0,C 180,E1 8356.119,E2 8356.119} C_VEL
LIN {X 0,Y 165.573,Z 1256.347,A -85,B 0,C 180,E1 8349.126,E2 8349.126} C_VEL
LIN {X 0,Y 170.424,Z 1250.969,A -85,B 0,C 180,E1 8342.364,E2 8342.364} C_VEL
LIN {X 0,Y 177.477,Z 1243.377,A -85,B 0,C 180,E1 8335.709,E2 8335.709} C_VEL
LIN {X 0,Y 186.017,Z 1234.053,A -85,B 0,C 180,E1 8329.832,E2 8329.832} C_VEL
LIN {X 0,Y 195.62,Z 1223.037,A -85,B 0,C 180,E1 8324.726,E2 8324.726} C_VEL
LIN {X 0,Y 205.288,Z 1211.092,A -85,B 0,C 180,E1 8320.552,E2 8320.552} C_VEL
LIN {X 0,Y 215.227,Z 1197.716,A -85,B 0,C 180,E1 8316.96,E2 8316.96} C_VEL
LIN {X 0,Y 219.122,Z 1191.983,A -85,B 0,C 180,E1 8315.638,E2 8315.638} C_VEL
LIN {X 0,Y 204.35,Z 1197.446,A -85,B 0,C 180,E1 8311.571,E2 8311.571} C_VEL
LIN {X 0,Y 194.252,Z 1200.928,A -85,B 0,C 180,E1 8307.931,E2 8307.931} C_VEL
LIN {X 0,Y 186.016,Z 1203.744,A -85,B 0,C 180,E1 8304.112,E2 8304.112} C_VEL
LIN {X 0,Y 179.094,Z 1206.156,A -85,B 0,C 180,E1 8299.911,E2 8299.911} C_VEL
LIN {X 0,Y 173.532,Z 1208.261,A -85,B 0,C 180,E1 8295.37,E2 8295.37} C_VEL
LIN {X 0,Y 169.491,Z 1210.102,A -85,B 0,C 180,E1 8290.882,E2 8290.882} C_VEL
LIN {X 0,Y 168.169,Z 1210.805,A -85,B 0,C 180,E1 8288.893,E2 8288.893} C_VEL
LIN {X 0,Y 166.147,Z 1212.204,A -85,B 0,C 180,E1 8284.834,E2 8284.834} C_VEL
LIN {X 0,Y 164.585,Z 1214.617,A -85,B 0,C 180,E1 8277.912,E2 8277.912} C_VEL
LIN {X 0,Y 164.799,Z 1215.256,A -85,B 0,C 180,E1 8276.522,E2 8276.522} C_VEL
LIN {X 0,Y 167.531,Z 1220.91,A -85,B 0,C 180,E1 8269.339,E2 8269.339} C_VEL
LIN {X 0,Y 172.403,Z 1224.627,A -85,B 0,C 180,E1 8262.448,E2 8262.448} C_VEL
LIN {X 0,Y 179.533,Z 1226.605,A -85,B 0,C 180,E1 8256.012,E2 8256.012} C_VEL
LIN {X 0,Y 190.404,Z 1226.888,A -85,B 0,C 180,E1 8249.379,E2 8249.379} C_VEL
LIN {X 0,Y 191.598,Z 1226.784,A -85,B 0,C 180,E1 8248.782,E2 8248.782} C_VEL
LIN {X 0,Y 193.188,Z 1227.063,A -85,B 0,C 180,E1 8247.504,E2 8247.504} C_VEL
LIN {X 0,Y 193.459,Z 1228.301,A -85,B 0,C 180,E1 8245.931,E2 8245.931} C_VEL
LIN {X 0,Y 192.326,Z 1230.624,A -85,B 0,C 180,E1 8244.171,E2 8244.171} C_VEL
LIN {X 0,Y 190.134,Z 1233.778,A -85,B 0,C 180,E1 8242.575,E2 8242.575} C_VEL
LIN {X 0,Y 189.081,Z 1235.19,A -85,B 0,C 180,E1 8242.054,E2 8242.054} C_VEL
LIN {X 0,Y 179.038,Z 1247.74,A -85,B 0,C 180,E1 8237.021,E2 8237.021} C_VEL
LIN {X 0,Y 170.481,Z 1258.099,A -85,B 0,C 180,E1 8231.511,E2 8231.511} C_VEL
LIN {X 0,Y 163.192,Z 1267.086,A -85,B 0,C 180,E1 8225.166,E2 8225.166} C_VEL
LIN {X 0,Y 157.614,Z 1274.603,A -85,B 0,C 180,E1 8217.999,E2 8217.999} C_VEL
LIN {X 0,Y 154.188,Z 1280.28,A -85,B 0,C 180,E1 8210.5,E2 8210.5} C_VEL
LIN {X 0,Y 152.743,Z 1284.206,A -85,B 0,C 180,E1 8202.861,E2 8202.861} C_VEL
LIN {X 0,Y 152.7,Z 1286.167,A -85,B 0,C 180,E1 8196.015,E2 8196.015} C_VEL
LIN {X 0,Y 152.893,Z 1286.791,A -85,B 0,C 180,E1 8190.376,E2 8190.376} C_VEL
LIN {X 0,Y 152.715,Z 1286.309,A -85,B 0,C 180,E1 8184.743,E2 8184.743} C_VEL
LIN {X 0,Y 152.606,Z 1284.701,A -85,B 0,C 180,E1 8178.666,E2 8178.666} C_VEL
LIN {X 0,Y 153.639,Z 1281.139,A -85,B 0,C 180,E1 8171.013,E2 8171.013} C_VEL
LIN {X 0,Y 156.586,Z 1275.841,A -85,B 0,C 180,E1 8163.452,E2 8163.452} C_VEL
LIN {X 0,Y 161.376,Z 1269.135,A -85,B 0,C 180,E1 8156.537,E2 8156.537} C_VEL
LIN {X 0,Y 168.528,Z 1260.094,A -85,B 0,C 180,E1 8149.71,E2 8149.71} C_VEL
LIN {X 0,Y 177.199,Z 1249.467,A -85,B 0,C 180,E1 8143.762,E2 8143.762} C_VEL
LIN {X 0,Y 186.446,Z 1237.885,A -85,B 0,C 180,E1 8138.86,E2 8138.86} C_VEL
LIN {X 0,Y 196.623,Z 1224.51,A -85,B 0,C 180,E1 8134.536,E2 8134.536} C_VEL
LIN {X 0,Y 207.255,Z 1209.44,A -85,B 0,C 180,E1 8130.829,E2 8130.829} C_VEL
LIN {X 0,Y 217.179,Z 1193.924,A -85,B 0,C 180,E1 8127.882,E2 8127.882} C_VEL
LIN {X 0,Y 226.451,Z 1177.778,A -85,B 0,C 180,E1 8125.495,E2 8125.495} C_VEL
LIN {X 0,Y 235.384,Z 1159.855,A -85,B 0,C 180,E1 8123.437,E2 8123.437} C_VEL
LIN {X 0,Y 242.926,Z 1142.196,A -85,B 0,C 180,E1 8121.858,E2 8121.858} C_VEL
LIN {X 0,Y 249.818,Z 1122.96,A -85,B 0,C 180,E1 8120.524,E2 8120.524} C_VEL
LIN {X 0,Y 255.453,Z 1103.37,A -85,B 0,C 180,E1 8119.498,E2 8119.498} C_VEL
LIN {X 0,Y 259.947,Z 1082.708,A -85,B 0,C 180,E1 8118.732,E2 8118.732} C_VEL
LIN {X 0,Y 262.98,Z 1061.014,A -85,B 0,C 180,E1 8118.155,E2 8118.155} C_VEL
LIN {X 0,Y 266.261,Z 1027.765,A -85,B 0,C 180,E1 8117.485,E2 8117.485} C_VEL
LIN {X 0,Y 269.516,Z 1000.127,A -85,B 0,C 180,E1 8117.282,E2 8117.282} C_VEL
LIN {X 0,Y 271.717,Z 983.081,A -85,B 0,C 180,E1 8117.287,E2 8117.287} C_VEL
LIN {X 0,Y 270.479,Z 964.237,A -85,B 0,C 180,E1 8114.668,E2 8114.668} C_VEL
LIN {X 0,Y 270.008,Z 943.523,A -85,B 0,C 180,E1 8111.995,E2 8111.995} C_VEL
LIN {X 0,Y 270.522,Z 919.086,A -85,B 0,C 180,E1 8109.233,E2 8109.233} C_VEL
LIN {X 0,Y 271.083,Z 906.817,A -85,B 0,C 180,E1 8107.95,E2 8107.95} C_VEL
LIN {X 0,Y 270.394,Z 900.304,A -85,B 0,C 180,E1 8105.41,E2 8105.41} C_VEL
LIN {X 0,Y 270.223,Z 891.643,A -85,B 0,C 180,E1 8101.59,E2 8101.59} C_VEL
LIN {X 0,Y 270.931,Z 885.046,A -85,B 0,C 180,E1 8098.308,E2 8098.308} C_VEL
LIN {X 0,Y 272.631,Z 878.582,A -85,B 0,C 180,E1 8094.739,E2 8094.739} C_VEL
LIN {X 0,Y 275.459,Z 872.604,A -85,B 0,C 180,E1 8091.02,E2 8091.02} C_VEL
LIN {X 0,Y 279.056,Z 867.931,A -85,B 0,C 180,E1 8087.585,E2 8087.585} C_VEL
LIN {X 0,Y 281.786,Z 865.926,A -85,B 0,C 180,E1 8085.408,E2 8085.408} C_VEL
LIN {X 0,Y 284.826,Z 873.227,A -85,B 0,C 180,E1 8082.533,E2 8082.533} C_VEL
LIN {X 0,Y 285.5,Z 875.136,A -85,B 0,C 180,E1 8081.941,E2 8081.941} C_VEL
LIN {X 0,Y 267.918,Z 1055.954,A -85,B 0,C 180,E1 8078.271,E2 8078.271} C_VEL
LIN {X 0,Y 264.571,Z 1076.419,A -85,B 0,C 180,E1 8077.598,E2 8077.598} C_VEL
LIN {X 0,Y 259.837,Z 1096.529,A -85,B 0,C 180,E1 8076.677,E2 8076.677} C_VEL
LIN {X 0,Y 253.83,Z 1115.988,A -85,B 0,C 180,E1 8075.492,E2 8075.492} C_VEL
LIN {X 0,Y 246.802,Z 1134.358,A -85,B 0,C 180,E1 8074.053,E2 8074.053} C_VEL
LIN {X 0,Y 238.444,Z 1152.554,A -85,B 0,C 180,E1 8072.222,E2 8072.222} C_VEL
LIN {X 0,Y 228.792,Z 1170.332,A -85,B 0,C 180,E1 8069.913,E2 8069.913} C_VEL
LIN {X 0,Y 218.796,Z 1186.275,A -85,B 0,C 180,E1 8067.227,E2 8067.227} C_VEL
LIN {X 0,Y 208.591,Z 1200.675,A -85,B 0,C 180,E1 8064.102,E2 8064.102} C_VEL
LIN {X 0,Y 198.379,Z 1213.651,A -85,B 0,C 180,E1 8060.454,E2 8060.454} C_VEL
LIN {X 0,Y 187.868,Z 1225.861,A -85,B 0,C 180,E1 8055.928,E2 8055.928} C_VEL
LIN {X 0,Y 178.268,Z 1236.219,A -85,B 0,C 180,E1 8050.783,E2 8050.783} C_VEL
LIN {X 0,Y 170.116,Z 1244.625,A -85,B 0,C 180,E1 8045.167,E2 8045.167} C_VEL
LIN {X 0,Y 163.037,Z 1251.799,A -85,B 0,C 180,E1 8038.576,E2 8038.576} C_VEL
LIN {X 0,Y 157.689,Z 1257.343,A -85,B 0,C 180,E1 8031.186,E2 8031.186} C_VEL
LIN {X 0,Y 154.571,Z 1260.881,A -85,B 0,C 180,E1 8023.846,E2 8023.846} C_VEL
LIN {X 0,Y 153.116,Z 1262.879,A -85,B 0,C 180,E1 8016.372,E2 8016.372} C_VEL
LIN {X 0,Y 152.821,Z 1263.463,A -85,B 0,C 180,E1 8009.623,E2 8009.623} C_VEL
LIN {X 0,Y 153.205,Z 1262.762,A -85,B 0,C 180,E1 8002.752,E2 8002.752} C_VEL
LIN {X 0,Y 154.769,Z 1260.649,A -85,B 0,C 180,E1 7995.405,E2 7995.405} C_VEL
LIN {X 0,Y 158.063,Z 1256.961,A -85,B 0,C 180,E1 7988.084,E2 7988.084} C_VEL
LIN {X 0,Y 163.285,Z 1251.604,A -85,B 0,C 180,E1 7981.068,E2 7981.068} C_VEL
LIN {X 0,Y 170.445,Z 1244.393,A -85,B 0,C 180,E1 7974.495,E2 7974.495} C_VEL
LIN {X 0,Y 178.925,Z 1235.657,A -85,B 0,C 180,E1 7968.744,E2 7968.744} C_VEL
LIN {X 0,Y 188.33,Z 1225.488,A -85,B 0,C 180,E1 7963.776,E2 7963.776} C_VEL
LIN {X 0,Y 198.662,Z 1213.474,A -85,B 0,C 180,E1 7959.358,E2 7959.358} C_VEL
LIN {X 0,Y 209.482,Z 1199.67,A -85,B 0,C 180,E1 7955.53,E2 7955.53} C_VEL
LIN {X 0,Y 209.613,Z 1199.378,A -85,B 0,C 180,E1 7955.42,E2 7955.42} C_VEL
LIN {X 0,Y 200.53,Z 1202.606,A -85,B 0,C 180,E1 7952.922,E2 7952.922} C_VEL
LIN {X 0,Y 190.091,Z 1206.06,A -85,B 0,C 180,E1 7949.287,E2 7949.287} C_VEL
LIN {X 0,Y 180.984,Z 1208.946,A -85,B 0,C 180,E1 7945.176,E2 7945.176} C_VEL
LIN {X 0,Y 173.769,Z 1211.297,A -85,B 0,C 180,E1 7940.901,E2 7940.901} C_VEL
LIN {X 0,Y 167.931,Z 1213.361,A -85,B 0,C 180,E1 7936.251,E2 7936.251} C_VEL
LIN {X 0,Y 163.473,Z 1215.254,A -85,B 0,C 180,E1 7931.288,E2 7931.288} C_VEL
LIN {X 0,Y 160.124,Z 1217.282,A -85,B 0,C 180,E1 7925.375,E2 7925.375} C_VEL
LIN {X 0,Y 158.452,Z 1219.772,A -85,B 0,C 180,E1 7917.831,E2 7917.831} C_VEL
LIN {X 0,Y 160.226,Z 1223.021,A -85,B 0,C 180,E1 7908.117,E2 7908.117} C_VEL
LIN {X 0,Y 162.162,Z 1224.342,A -85,B 0,C 180,E1 7904.992,E2 7904.992} C_VEL
LIN {X 0,Y 168.561,Z 1227.533,A -85,B 0,C 180,E1 7898.057,E2 7898.057} C_VEL
LIN {X 0,Y 177.809,Z 1229.129,A -85,B 0,C 180,E1 7891.448,E2 7891.448} C_VEL
LIN {X 0,Y 193.467,Z 1229.168,A -85,B 0,C 180,E1 7884.086,E2 7884.086} C_VEL
LIN {X 0,Y 193.436,Z 1229.514,A -85,B 0,C 180,E1 7883.896,E2 7883.896} C_VEL
LIN {X 0,Y 189.081,Z 1235.19,A -85,B 0,C 180,E1 7882.054,E2 7882.054} C_VEL
LIN {X 0,Y 184.829,Z 1239.778,A -85,B 0,C 180,E1 7880.64,E2 7880.64} C_VEL
LIN {X 0,Y 171.401,Z 1250.444,A -85,B 0,C 180,E1 7877.241,E2 7877.241} C_VEL
LIN {X 0,Y 167.262,Z 1254.18,A -85,B 0,C 180,E1 7875.411,E2 7875.411} C_VEL
LIN {X 0,Y 158.742,Z 1263.875,A -85,B 0,C 180,E1 7869.042,E2 7869.042} C_VEL
LIN {X 0,Y 151.937,Z 1271.947,A -85,B 0,C 180,E1 7861.768,E2 7861.768} C_VEL
LIN {X 0,Y 147.411,Z 1278.129,A -85,B 0,C 180,E1 7854.016,E2 7854.016} C_VEL
LIN {X 0,Y 145.101,Z 1282.539,A -85,B 0,C 180,E1 7846.001,E2 7846.001} C_VEL
LIN {X 0,Y 144.623,Z 1285.099,A -85,B 0,C 180,E1 7838.652,E2 7838.652} C_VEL
LIN {X 0,Y 144.853,Z 1286.029,A -85,B 0,C 180,E1 7832.771,E2 7832.771} C_VEL
LIN {X 0,Y 144.879,Z 1286.079,A -85,B 0,C 180,E1 7828.024,E2 7828.024} C_VEL
LIN {X 0,Y 144.632,Z 1285.306,A -85,B 0,C 180,E1 7822.454,E2 7822.454} C_VEL
LIN {X 0,Y 144.913,Z 1282.86,A -85,B 0,C 180,E1 7814.802,E2 7814.802} C_VEL
LIN {X 0,Y 146.791,Z 1278.901,A -85,B 0,C 180,E1 7807.156,E2 7807.156} C_VEL
LIN {X 0,Y 151.192,Z 1272.616,A -85,B 0,C 180,E1 7798.949,E2 7798.949} C_VEL
LIN {X 0,Y 157.72,Z 1264.665,A -85,B 0,C 180,E1 7791.594,E2 7791.594} C_VEL
LIN {X 0,Y 165.926,Z 1255.208,A -85,B 0,C 180,E1 7785.17,E2 7785.17} C_VEL
LIN {X 0,Y 175.341,Z 1244.337,A -85,B 0,C 180,E1 7779.665,E2 7779.665} C_VEL
LIN {X 0,Y 186.175,Z 1231.324,A -85,B 0,C 180,E1 7774.748,E2 7774.748} C_VEL
LIN {X 0,Y 197.133,Z 1217.136,A -85,B 0,C 180,E1 7770.72,E2 7770.72} C_VEL
LIN {X 0,Y 207.849,Z 1201.931,A -85,B 0,C 180,E1 7767.438,E2 7767.438} C_VEL
LIN {X 0,Y 218.009,Z 1185.857,A -85,B 0,C 180,E1 7764.761,E2 7764.761} C_VEL
LIN {X 0,Y 227.822,Z 1168.172,A -85,B 0,C 180,E1 7762.51,E2 7762.51} C_VEL
LIN {X 0,Y 236.712,Z 1149.447,A -85,B 0,C 180,E1 7760.678,E2 7760.678} C_VEL
LIN {X 0,Y 244.158,Z 1130.804,A -85,B 0,C 180,E1 7759.282,E2 7759.282} C_VEL
LIN {X 0,Y 250.468,Z 1111.522,A -85,B 0,C 180,E1 7758.183,E2 7758.183} C_VEL
LIN {X 0,Y 255.509,Z 1091.734,A -85,B 0,C 180,E1 7757.34,E2 7757.34} C_VEL
LIN {X 0,Y 259.314,Z 1070.825,A -85,B 0,C 180,E1 7756.721,E2 7756.721} C_VEL
LIN {X 0,Y 263.711,Z 1029.529,A -85,B 0,C 180,E1 7755.852,E2 7755.852} C_VEL
LIN {X 0,Y 267.07,Z 1001.065,A -85,B 0,C 180,E1 7755.647,E2 7755.647} C_VEL
LIN {X 0,Y 269.081,Z 985.375,A -85,B 0,C 180,E1 7755.653,E2 7755.653} C_VEL
LIN {X 0,Y 268.257,Z 966.566,A -85,B 0,C 180,E1 7753.059,E2 7753.059} C_VEL
LIN {X 0,Y 268.12,Z 947.716,A -85,B 0,C 180,E1 7750.596,E2 7750.596} C_VEL
LIN {X 0,Y 268.988,Z 922.496,A -85,B 0,C 180,E1 7747.73,E2 7747.73} C_VEL
LIN {X 0,Y 269.558,Z 912.445,A -85,B 0,C 180,E1 7746.656,E2 7746.656} C_VEL
LIN {X 0,Y 269.171,Z 907.216,A -85,B 0,C 180,E1 7744.58,E2 7744.58} C_VEL
LIN {X 0,Y 269.245,Z 898.793,A -85,B 0,C 180,E1 7740.851,E2 7740.851} C_VEL
LIN {X 0,Y 270.15,Z 892.231,A -85,B 0,C 180,E1 7737.56,E2 7737.56} C_VEL
LIN {X 0,Y 272.07,Z 885.761,A -85,B 0,C 180,E1 7733.987,E2 7733.987} C_VEL
LIN {X 0,Y 275.419,Z 879.456,A -85,B 0,C 180,E1 7729.964,E2 7729.964} C_VEL
LIN {X 0,Y 278.794,Z 875.453,A -85,B 0,C 180,E1 7726.941,E2 7726.941} C_VEL
LIN {X 0,Y 280.608,Z 874.293,A -85,B 0,C 180,E1 7725.503,E2 7725.503} C_VEL
LIN {X 0,Y 282.7,Z 879.858,A -85,B 0,C 180,E1 7723.397,E2 7723.397} C_VEL
LIN {X 0,Y 265.054,Z 1056.577,A -85,B 0,C 180,E1 7719.871,E2 7719.871} C_VEL
LIN {X 0,Y 261.621,Z 1077.039,A -85,B 0,C 180,E1 7719.212,E2 7719.212} C_VEL
LIN {X 0,Y 256.799,Z 1097.042,A -85,B 0,C 180,E1 7718.317,E2 7718.317} C_VEL
LIN {X 0,Y 250.621,Z 1116.577,A -85,B 0,C 180,E1 7717.155,E2 7717.155} C_VEL
LIN {X 0,Y 243.409,Z 1134.954,A -85,B 0,C 180,E1 7715.746,E2 7715.746} C_VEL
LIN {X 0,Y 234.818,Z 1153.155,A -85,B 0,C 180,E1 7713.951,E2 7713.951} C_VEL
LIN {X 0,Y 224.876,Z 1170.937,A -85,B 0,C 180,E1 7711.683,E2 7711.683} C_VEL
LIN {X 0,Y 214.551,Z 1186.883,A -85,B 0,C 180,E1 7709.032,E2 7709.032} C_VEL
LIN {X 0,Y 203.974,Z 1201.286,A -85,B 0,C 180,E1 7705.934,E2 7705.934} C_VEL
LIN {X 0,Y 193.344,Z 1214.265,A -85,B 0,C 180,E1 7702.298,E2 7702.298} C_VEL
LIN {X 0,Y 182.342,Z 1226.476,A -85,B 0,C 180,E1 7697.751,E2 7697.751} C_VEL
LIN {X 0,Y 172.498,Z 1236.571,A -85,B 0,C 180,E1 7692.699,E2 7692.699} C_VEL
LIN {X 0,Y 163.552,Z 1245.258,A -85,B 0,C 180,E1 7686.787,E2 7686.787} C_VEL
LIN {X 0,Y 155.986,Z 1252.416,A -85,B 0,C 180,E1 7679.996,E2 7679.996} C_VEL
LIN {X 0,Y 150.181,Z 1257.978,A -85,B 0,C 180,E1 7672.266,E2 7672.266} C_VEL
LIN {X 0,Y 146.779,Z 1261.495,A -85,B 0,C 180,E1 7664.597,E2 7664.597} C_VEL
LIN {X 0,Y 145.172,Z 1263.489,A -85,B 0,C 180,E1 7656.722,E2 7656.722} C_VEL
LIN {X 0,Y 144.844,Z 1264.071,A -85,B 0,C 180,E1 7649.603,E2 7649.603} C_VEL
LIN {X 0,Y 145.255,Z 1263.393,A -85,B 0,C 180,E1 7642.483,E2 7642.483} C_VEL
LIN {X 0,Y 147.004,Z 1261.262,A -85,B 0,C 180,E1 7634.616,E2 7634.616} C_VEL
LIN {X 0,Y 150.606,Z 1257.576,A -85,B 0,C 180,E1 7626.938,E2 7626.938} C_VEL
LIN {X 0,Y 156.257,Z 1252.219,A -85,B 0,C 180,E1 7619.633,E2 7619.633} C_VEL
LIN {X 0,Y 163.926,Z 1245.008,A -85,B 0,C 180,E1 7612.852,E2 7612.852} C_VEL
LIN {X 0,Y 172.926,Z 1236.27,A -85,B 0,C 180,E1 7606.977,E2 7606.977} C_VEL
LIN {X 0,Y 182.832,Z 1226.099,A -85,B 0,C 180,E1 7601.947,E2 7601.947} C_VEL
LIN {X 0,Y 193.465,Z 1214.292,A -85,B 0,C 180,E1 7597.579,E2 7597.579} C_VEL
LIN {X 0,Y 199.88,Z 1206.594,A -85,B 0,C 180,E1 7595.295,E2 7595.295} C_VEL
LIN {X 0,Y 185.877,Z 1210.963,A -85,B 0,C 180,E1 7590.732,E2 7590.732} C_VEL
LIN {X 0,Y 175.897,Z 1213.988,A -85,B 0,C 180,E1 7586.32,E2 7586.32} C_VEL
LIN {X 0,Y 168.377,Z 1216.277,A -85,B 0,C 180,E1 7581.97,E2 7581.97} C_VEL
LIN {X 0,Y 162.129,Z 1218.33,A -85,B 0,C 180,E1 7577.076,E2 7577.076} C_VEL
LIN {X 0,Y 157.536,Z 1220.153,A -85,B 0,C 180,E1 7572.091,E2 7572.091} C_VEL
LIN {X 0,Y 153.948,Z 1222.144,A -85,B 0,C 180,E1 7565.966,E2 7565.966} C_VEL
LIN {X 0,Y 152.085,Z 1224.579,A -85,B 0,C 180,E1 7558.117,E2 7558.117} C_VEL
LIN {X 0,Y 153.997,Z 1227.903,A -85,B 0,C 180,E1 7547.629,E2 7547.629} C_VEL
LIN {X 0,Y 163.862,Z 1231.56,A -85,B 0,C 180,E1 7535.486,E2 7535.486} C_VEL
LIN {X 0,Y 178.139,Z 1233.495,A -85,B 0,C 180,E1 7527.014,E2 7527.014} C_VEL
LIN {X 0,Y 184.624,Z 1233.873,A -85,B 0,C 180,E1 7524.328,E2 7524.328} C_VEL
LIN {X 0,Y 174.554,Z 1245.795,A -85,B 0,C 180,E1 7519.628,E2 7519.628} C_VEL
LIN {X 0,Y 167.262,Z 1254.18,A -85,B 0,C 180,E1 7515.411,E2 7515.411} C_VEL
LIN {X 0,Y 163.234,Z 1257.781,A -85,B 0,C 180,E1 7513.461,E2 7513.461} C_VEL
LIN {X 0,Y 150.637,Z 1265.984,A -85,B 0,C 180,E1 7508.57,E2 7508.57} C_VEL
LIN {X 0,Y 147.162,Z 1268.783,A -85,B 0,C 180,E1 7506.123,E2 7506.123} C_VEL
LIN {X 0,Y 141.368,Z 1275.579,A -85,B 0,C 180,E1 7498.288,E2 7498.288} C_VEL
LIN {X 0,Y 137.908,Z 1280.596,A -85,B 0,C 180,E1 7489.925,E2 7489.925} C_VEL
LIN {X 0,Y 136.692,Z 1283.737,A -85,B 0,C 180,E1 7481.82,E2 7481.82} C_VEL
LIN {X 0,Y 136.79,Z 1285.302,A -85,B 0,C 180,E1 7474.614,E2 7474.614} C_VEL
LIN {X 0,Y 136.929,Z 1285.546,A -85,B 0,C 180,E1 7469.165,E2 7469.165} C_VEL
LIN {X 0,Y 136.678,Z 1284.926,A -85,B 0,C 180,E1 7463.28,E2 7463.28} C_VEL
LIN {X 0,Y 136.785,Z 1283.072,A -85,B 0,C 180,E1 7456.043,E2 7456.043} C_VEL
LIN {X 0,Y 138.444,Z 1279.432,A -85,B 0,C 180,E1 7447.944,E2 7447.944} C_VEL
LIN {X 0,Y 142.449,Z 1273.927,A -85,B 0,C 180,E1 7439.646,E2 7439.646} C_VEL
LIN {X 0,Y 148.952,Z 1266.491,A -85,B 0,C 180,E1 7431.754,E2 7431.754} C_VEL
LIN {X 0,Y 157.096,Z 1257.788,A -85,B 0,C 180,E1 7425.054,E2 7425.054} C_VEL
LIN {X 0,Y 167.202,Z 1246.984,A -85,B 0,C 180,E1 7418.98,E2 7418.98} C_VEL
LIN {X 0,Y 178.265,Z 1234.6,A -85,B 0,C 180,E1 7413.893,E2 7413.893} C_VEL
LIN {X 0,Y 189.52,Z 1220.993,A -85,B 0,C 180,E1 7409.73,E2 7409.73} C_VEL
LIN {X 0,Y 200.749,Z 1206.116,A -85,B 0,C 180,E1 7406.3,E2 7406.3} C_VEL
LIN {X 0,Y 211.514,Z 1190.207,A -85,B 0,C 180,E1 7403.503,E2 7403.503} C_VEL
LIN {X 0,Y 221.938,Z 1172.747,A -85,B 0,C 180,E1 7401.166,E2 7401.166} C_VEL
LIN {X 0,Y 231.015,Z 1155.171,A -85,B 0,C 180,E1 7399.351,E2 7399.351} C_VEL
LIN {X 0,Y 239.157,Z 1136.639,A -85,B 0,C 180,E1 7397.877,E2 7397.877} C_VEL
LIN {X 0,Y 246.317,Z 1116.653,A -85,B 0,C 180,E1 7396.674,E2 7396.674} C_VEL
LIN {X 0,Y 251.869,Z 1096.93,A -85,B 0,C 180,E1 7395.809,E2 7395.809} C_VEL
LIN {X 0,Y 256.161,Z 1076.054,A -85,B 0,C 180,E1 7395.142,E2 7395.142} C_VEL
LIN {X 0,Y 259.405,Z 1050.275,A -85,B 0,C 180,E1 7394.55,E2 7394.55} C_VEL
LIN {X 0,Y 262.354,Z 1022.627,A -85,B 0,C 180,E1 7394.085,E2 7394.085} C_VEL
LIN {X 0,Y 266.309,Z 990.642,A -85,B 0,C 180,E1 7394.003,E2 7394.003} C_VEL
LIN {X 0,Y 266.663,Z 987.44,A -85,B 0,C 180,E1 7393.96,E2 7393.96} C_VEL
LIN {X 0,Y 266.287,Z 955.971,A -85,B 0,C 180,E1 7389.673,E2 7389.673} C_VEL
LIN {X 0,Y 267.577,Z 926.878,A -85,B 0,C 180,E1 7386.309,E2 7386.309} C_VEL
LIN {X 0,Y 268.186,Z 918.188,A -85,B 0,C 180,E1 7385.407,E2 7385.407} C_VEL
LIN {X 0,Y 267.989,Z 913.541,A -85,B 0,C 180,E1 7383.475,E2 7383.475} C_VEL
LIN {X 0,Y 268.312,Z 905.946,A -85,B 0,C 180,E1 7380.106,E2 7380.106} C_VEL
LIN {X 0,Y 269.37,Z 899.594,A -85,B 0,C 180,E1 7376.914,E2 7376.914} C_VEL
LIN {X 0,Y 272.209,Z 891.46,A -85,B 0,C 180,E1 7372.401,E2 7372.401} C_VEL
LIN {X 0,Y 277.211,Z 884.192,A -85,B 0,C 180,E1 7367.395,E2 7367.395} C_VEL
LIN {X 0,Y 279.329,Z 882.497,A -85,B 0,C 180,E1 7365.7,E2 7365.7} C_VEL
LIN {X 0,Y 280.065,Z 884.768,A -85,B 0,C 180,E1 7364.877,E2 7364.877} C_VEL
LIN {X 0,Y 262.401,Z 1057.198,A -85,B 0,C 180,E1 7361.506,E2 7361.506} C_VEL
LIN {X 0,Y 258.894,Z 1077.607,A -85,B 0,C 180,E1 7360.863,E2 7360.863} C_VEL
LIN {X 0,Y 253.977,Z 1097.552,A -85,B 0,C 180,E1 7359.994,E2 7359.994} C_VEL
LIN {X 0,Y 248.042,Z 1116.063,A -85,B 0,C 180,E1 7358.932,E2 7358.932} C_VEL
LIN {X 0,Y 240.675,Z 1134.597,A -85,B 0,C 180,E1 7357.568,E2 7357.568} C_VEL
LIN {X 0,Y 231.75,Z 1153.098,A -85,B 0,C 180,E1 7355.803,E2 7355.803} C_VEL
LIN {X 0,Y 221.954,Z 1170.241,A -85,B 0,C 180,E1 7353.693,E2 7353.693} C_VEL
LIN {X 0,Y 211.566,Z 1185.987,A -85,B 0,C 180,E1 7351.18,E2 7351.18} C_VEL
LIN {X 0,Y 201.003,Z 1200.098,A -85,B 0,C 180,E1 7348.275,E2 7348.275} C_VEL
LIN {X 0,Y 189.864,Z 1213.385,A -85,B 0,C 180,E1 7344.709,E2 7344.709} C_VEL
LIN {X 0,Y 178.854,Z 1225.252,A -85,B 0,C 180,E1 7340.483,E2 7340.483} C_VEL
LIN {X 0,Y 168.291,Z 1235.692,A -85,B 0,C 180,E1 7335.473,E2 7335.473} C_VEL
LIN {X 0,Y 158.09,Z 1245.054,A -85,B 0,C 180,E1 7329.23,E2 7329.23} C_VEL
LIN {X 0,Y 149.756,Z 1252.37,A -85,B 0,C 180,E1 7322.283,E2 7322.283} C_VEL
LIN {X 0,Y 143.512,Z 1257.856,A -85,B 0,C 180,E1 7314.708,E2 7314.708} C_VEL
LIN {X 0,Y 139.446,Z 1261.664,A -85,B 0,C 180,E1 7306.665,E2 7306.665} C_VEL
LIN {X 0,Y 137.393,Z 1263.915,A -85,B 0,C 180,E1 7298.367,E2 7298.367} C_VEL
LIN {X 0,Y 136.871,Z 1264.628,A -85,B 0,C 180,E1 7291.254,E2 7291.254} C_VEL
LIN {X 0,Y 137.138,Z 1264.25,A -85,B 0,C 180,E1 7283.72,E2 7283.72} C_VEL
LIN {X 0,Y 138.617,Z 1262.605,A -85,B 0,C 180,E1 7275.802,E2 7275.802} C_VEL
LIN {X 0,Y 142.255,Z 1259.075,A -85,B 0,C 180,E1 7267.257,E2 7267.257} C_VEL
LIN {X 0,Y 147.937,Z 1254.007,A -85,B 0,C 180,E1 7259.541,E2 7259.541} C_VEL
LIN {X 0,Y 155.744,Z 1247.167,A -85,B 0,C 180,E1 7252.417,E2 7252.417} C_VEL
LIN {X 0,Y 165.557,Z 1238.302,A -85,B 0,C 180,E1 7245.947,E2 7245.947} C_VEL
LIN {X 0,Y 176.315,Z 1227.937,A -85,B 0,C 180,E1 7240.543,E2 7240.543} C_VEL
LIN {X 0,Y 187.097,Z 1216.649,A -85,B 0,C 180,E1 7236.199,E2 7236.199} C_VEL
